# B&R Automation Studio project A2019059_Linka_Power_CP (part 37)

#### Main.st - Init, cyclic, exit code
```iecst
PROGRAM _INIT
    TprazdnyZasobnik.PT:=T#2000ms;
    TakumulaciaPlna.PT:=T#1000ms;
    TvytvorenieVakua.PT:=T#200ms;
    TodvetranieVakua.PT:=T#1s;
    TprefukPredBrzdou.PT:=T#2000ms;
    TprefukZaBrzdou.PT:=T#2000ms;
    TvysuvanieSpindle.PT:=T#1s;
    TpripravaSkrutky.PT:=T#3000ms;
    ToddelovacZakladnaPoloha.PT:=T#1000ms;
    TodsatieNecistot.PT:=T#1000ms;
    Tvibrovanie.PT:=T#3000ms;
    TvyfukovaniePredVibrovanim.PT:= T#1000ms;
    TpodaniaSkrutky.PT:= T#1000ms;
    TpredSkrutkaPripravena.PT:= T#1000ms;
    TvypnutieOfuku.PT:= T#2000ms;
    TalarmuVysunutiaSkrutkovacky.PT:= T#10s;
END_PROGRAM

PROGRAM _CYCLIC

	(********************Mapovanie IN/OUT********************************)

    SkrutkovaciSet.Manual:= P3_Srobovanie.SkrutkovaciSet_K40.Manual;
    SkrutkovaciSet.Automat:= P3_Srobovanie.SkrutkovaciSet_K40.Automat;
    SkrutkovaciSet.SkrutkaOdobrata:=P3_Srobovanie.SkrutkovaciSet_K40.SkrutkaK40_Odobrata;
    P3_Srobovanie.SkrutkovaciSet_K40.SkrutkaK40_Pripravena:= SkrutkovaciSet.SkrutkaPripravena;
    P3_Srobovanie.SkrutkovaciSet_K40.CistenieUkoncene:= SkrutkovaciSet.CistenieVykonane;
    SkrutkovaciSet.VykonajCistenie:= P3_Srobovanie.SkrutkovaciSet_K40.Cistenie;

    SkrutkovaciSet.Vreteno.IN.BrakeClosed:=P3_Srobovanie.IN.SkrutkK40_Cist_BrzdaZatvor_MS54;
    SkrutkovaciSet.Vreteno.IN.BrakeOpen:=P3_Srobovanie.IN.SkrutkK40_Cist_BrzdaOtvor_MS53;
    SkrutkovaciSet.Vreteno.IN.DeptControl:=P3_Srobovanie.IN.SkrutkK40_ZASUNUTY_MS52;
    SkrutkovaciSet.Vreteno.IN.ScrewMeasurement:=P3_Srobovanie.IN.SkrutkK40_SrobaPresla_IS81;
    SkrutkovaciSet.Vreteno.IN.ScrewMeasurementBrake:=P3_Srobovanie.IN.SkrutkK40_Cist_SrobaPresla_IS82;

    IF P3_Srobovanie.SkrutkovaciSet_K40.Reset AND SkrutkovaciSet.VretenoFaza <> 102 AND SkrutkovaciSet.VretenoFaza <> 104 THEN
        SkrutkovaciSet.VretenoFaza:=0;
        P3_Srobovanie.SkrutkovaciSet_K40.Reset:= FALSE;
    END_IF

    SkrutkovaciSet.Zasobnik.IN.AccumulationSwitch:=P3_Srobovanie.IN.ZasobSrobK40_ListaPLNA_OS15;
    SkrutkovaciSet.Zasobnik.IN.FeederLevelControl:=P3_Srobovanie.IN.ZasobSrobK40_PRAZDNY_IS79;
    SkrutkovaciSet.Zasobnik.IN.ScrewMeasurement:=P3_Srobovanie.IN.NastrelSrobK40_SrobaPresla_IS80;

    P3_Srobovanie.OUT.SkrutkK40_Cist_POSUN_YV124:=SkrutkovaciSet.Vreteno.OUT.BlastAirBrake;
    P3_Srobovanie.OUT.SkrutkK40_Cist_OTVOR_YV121:=SkrutkovaciSet.Vreteno.OUT.BrakeSpindle;
    P3_Srobovanie.OUT.SkrutkK40_OfukVakua_RUN_YV119:=SkrutkovaciSet.Vreteno.OUT.CounterBlast;
    IF SkrutkovaciSet.VretenoFaza>1 AND SkrutkovaciSet.VretenoFaza<100 THEN
        P3_Srobovanie.OUT.SkrutkK40_VYSUN_YV118:=SkrutkovaciSet.Vreteno.OUT.Spindle;
    END_IF
    P3_Srobovanie.OUT.SkrutkK40_Cist_ODSAVANIE_YV122:=SkrutkovaciSet.Vreteno.OUT.WasteExtraction;
    IF SkrutkovaciSet.VykonajCistenie THEN
        P3_Srobovanie.OUT.SkrutkK40_PrisavSkrut_RUN_YV120:=SkrutkovaciSet.Vreteno.OUT.Vacuum;
    END_IF
    P3_Srobovanie.OUT.ZasobSrobK40_Ofuk_RUN_YV114:=SkrutkovaciSet.Zasobnik.OUT.BlowOff;
    P3_Srobovanie.OUT.NastrelSrobK40_PosunSrobu_YV116:=SkrutkovaciSet.Zasobnik.OUT.Escapement;
    P3_Srobovanie.OUT.NastrelSrobK40_NastrelSrob_YV117:=SkrutkovaciSet.Zasobnik.OUT.FeedAir;
    P3_Srobovanie.OUT.ZasobSrobK40_OfukTried_RUN_YV115:=SkrutkovaciSet.Zasobnik.OUT.SortingAir;
    P3_Srobovanie.OUT.ZasobSrobK40_Vibrovanie_RUN_FM15:= SkrutkovaciSet.Zasobnik.OUT.StartA20;
    (********************Časáky********************************)
    TprazdnyZasobnik();
    TakumulaciaPlna();
    TvytvorenieVakua();
    TodvetranieVakua();
    TprefukPredBrzdou();
    TprefukZaBrzdou();
    TvysuvanieSpindle();
    TpripravaSkrutky();
    ToddelovacZakladnaPoloha();
    TodsatieNecistot();
    Tvibrovanie();
    TvyfukovaniePredVibrovanim();
    TpodaniaSkrutky();
    TpredSkrutkaPripravena();
    TvypnutieOfuku();
    TalarmuVysunutiaSkrutkovacky();
    (********************Zásobnik********************************)

    //kontrola akumulacie
    IF SkrutkovaciSet.Zasobnik.IN.AccumulationSwitch=1 THEN
        TakumulaciaPlna.IN:=1;
    ELSE
        TakumulaciaPlna.IN:=0;
    END_IF

    //kontrola naplnenia zasobnika
    IF SkrutkovaciSet.Zasobnik.IN.FeederLevelControl=1 THEN
        TprazdnyZasobnik.IN:=1;
    ELSE
        TprazdnyZasobnik.IN:=0;
    END_IF

    //Ovládanie vzduchov zásobníka//
    IF ZapniHrniec THEN
        IF TakumulaciaPlna.Q=1 THEN
            SkrutkovaciSet.Zasobnik.OUT.BlowOff:=1;
        ELSE
            SkrutkovaciSet.Zasobnik.OUT.BlowOff:=0;
        END_IF
        SkrutkovaciSet.Zasobnik.OUT.SortingAir:= 1;
    ELSE
        SkrutkovaciSet.Zasobnik.OUT.BlowOff:=0;
    END_IF

    IF NOT SkrutkovaciSet.Zasobnik.OUT.StartA20 AND NOT ZapniHrniec THEN
        TvypnutieOfuku.IN:= 1;
    ELSE
        TvypnutieOfuku.IN:= 0;
    END_IF

    IF EDGEPOS(TvypnutieOfuku.Q) THEN
        SkrutkovaciSet.Zasobnik.OUT.SortingAir:= 0;
    END_IF

    //ovladanie vibracneho podavaca
    IF ZapniHrniec THEN
        TvyfukovaniePredVibrovanim.IN:= 1;
    ELSE
        TvyfukovaniePredVibrovanim.IN:= 0;
    END_IF

    IF ZapniHrniec AND TvyfukovaniePredVibrovanim.Q THEN
        SkrutkovaciSet.Zasobnik.OUT.StartA20:=1;
        Tvibrovanie.IN:=1;
    ELSE
        SkrutkovaciSet.Zasobnik.OUT.StartA20:=0;
        Tvibrovanie.IN:=0;
    END_IF

    IF Tvibrovanie.Q=1 AND NOT P3_Srobovanie.RR_ZapniHrniec_K40 THEN
        IF TakumulaciaPlna.Q=1 THEN
            ZapniHrniec:= 0;
        END_IF
    END_IF

    //Zapnutie hrnca v ručnom režime//
    IF EDGEPOS(P3_Srobovanie.RR_ZapniHrniec_K40) THEN
        ZapniHrniec:= TRUE;
    END_IF
    IF EDGENEG(P3_Srobovanie.RR_ZapniHrniec_K40) THEN
        ZapniHrniec:= FALSE;
    END_IF

    //Zrušenie signálu skrutka pripravená//
    IF SkrutkovaciSet.SkrutkaPripravena=1 THEN
        IF SkrutkovaciSet.SkrutkaOdobrata=1 THEN
            SkrutkovaciSet.SkrutkaPripravena:=0;
        END_IF
    END_IF

    (********************Vreteno********************************)
    CASE SkrutkovaciSet.VretenoFaza OF
        0: SkrutkovaciSet.VretenoStatus:="Vypnute";
            SkrutkovaciSet.Vreteno.OUT.BlastAirBrake:=0;
            SkrutkovaciSet.Vreteno.OUT.BrakeSpindle:=0;
            SkrutkovaciSet.Vreteno.OUT.CounterBlast:=0;
            SkrutkovaciSet.Vreteno.OUT.Spindle:=0;
            SkrutkovaciSet.Vreteno.OUT.Vacuum:=0;
            SkrutkovaciSet.Vreteno.OUT.WasteExtraction:=0;

            SkrutkovaciSet.Zasobnik.OUT.Escapement:=0;
            SkrutkovaciSet.Zasobnik.OUT.FeedAir:=0;

            SkrutkovaciSet.Zasobnik.OUT.StartA20:=0;

            SkrutkovaciSet.CistenieVykonane:=0;
            SkrutkovaciSet.SkrutkaPripravena:=0;

            TprazdnyZasobnik.IN:=0;
            TakumulaciaPlna.IN:=0;
            TvytvorenieVakua.IN:=0;
            TodvetranieVakua.IN:=0;
            TprefukPredBrzdou.IN:=0;
            TprefukZaBrzdou.IN:=0;
            TvysuvanieSpindle.IN:=0;
            TpripravaSkrutky.IN:=0;
            ToddelovacZakladnaPoloha.IN:=0;
            TodsatieNecistot.IN:=0;
            TpodaniaSkrutky.IN:= 0;
            TpredSkrutkaPripravena.IN:= 0;
            ZapniHrniec:= 0;
            PocetPokusovOpripravuSkrutky:=0;
            TalarmuVysunutiaSkrutkovacky.IN:= 0;
            StavSkrutkovackaVysunuta:= 0;
            SkrutkovaciSet.VretenoFaza:=1;

        1: SkrutkovaciSet.VretenoStatus:="Inicializacia: cakam na povel";
            IF SkrutkovaciSet.Automat=1 THEN
                SkrutkovaciSet.CistenieVykonane:=0;
                SkrutkovaciSet.SkrutkaPripravena:=0;
                SkrutkovaciSet.VretenoFaza:=2;
            ELSIF SkrutkovaciSet.Manual=1 THEN
                SkrutkovaciSet.VretenoFaza:=250;
            END_IF

        2: SkrutkovaciSet.VretenoStatus:="Inicializacia: cakam na povel precisti hadice";

            IF SkrutkovaciSet.VykonajCistenie=1 THEN
                SkrutkovaciSet.Vreteno.OUT.Vacuum:=1;
                SkrutkovaciSet.VretenoFaza:=3;
            END_IF

        3: SkrutkovaciSet.VretenoStatus:="Inicializacia: Cakam na snimac: vreteno vysunute";
            SkrutkovaciSet.Vreteno.OUT.Spindle:=1;
            TalarmuVysunutiaSkrutkovacky.IN:= 1;

            IF P3_Srobovanie.IN.SkrutkK40_VysunutieHrotu_IOS11 > 1 THEN
                StavSkrutkovackaVysunuta:= TRUE;
                TvysuvanieSpindle.IN:=1;
            END_IF

            IF TvysuvanieSpindle.Q=1 AND StavSkrutkovackaVysunuta THEN
                TodvetranieVakua.IN:= 1;
                SkrutkovaciSet.Vreteno.OUT.CounterBlast:=1;
                SkrutkovaciSet.Vreteno.OUT.Vacuum:=0;
            END_IF

            IF TvysuvanieSpindle.Q AND StavSkrutkovackaVysunuta AND TodvetranieVakua.Q THEN
                StavSkrutkovackaVysunuta:= FALSE;
                TalarmuVysunutiaSkrutkovacky.IN:= 0;
                TvysuvanieSpindle.IN:=0;
                TodvetranieVakua.IN:= 0;
                SkrutkovaciSet.VretenoFaza:=4;
            ELSIF TalarmuVysunutiaSkrutkovacky.Q THEN
                P34_Alarmy[342]:= TRUE;
                P3_PoruchaST1:= TRUE;
            END_IF

        4: SkrutkovaciSet.VretenoStatus:="Inicializacia: Cakam na snimac: vreteno zasunute";
            SkrutkovaciSet.Vreteno.OUT.Spindle:=0;
            IF SkrutkovaciSet.Vreteno.IN.DeptControl=1 THEN
                SkrutkovaciSet.Vreteno.OUT.CounterBlast:=0;
                SkrutkovaciSet.VretenoFaza:=5;
            END_IF

        5: SkrutkovaciSet.VretenoStatus:="Inicializacia: Cakam na prefuknutie hadice za brzdou";
            TprefukZaBrzdou.IN:=1;
            SkrutkovaciSet.Vreteno.OUT.BlastAirBrake:=1;
            IF TprefukZaBrzdou.Q=1 THEN
                TprefukZaBrzdou.IN:=0;
                SkrutkovaciSet.Vreteno.OUT.BlastAirBrake:=0;
                SkrutkovaciSet.VretenoFaza:=6;
            END_IF

        6: SkrutkovaciSet.VretenoStatus:="Inicializacia: vypinam prefuk";
            TprefukZaBrzdou.IN:=0;
            SkrutkovaciSet.Vreteno.OUT.BlastAirBrake:=0;
            SkrutkovaciSet.Vreteno.OUT.Vacuum:=1;
            SkrutkovaciSet.VretenoFaza:=7;

        7: SkrutkovaciSet.VretenoStatus:="Inicializacia: Cakam na snimac: vreteno vysunute";
            SkrutkovaciSet.Vreteno.OUT.Spindle:=1;
            TalarmuVysunutiaSkrutkovacky.IN:= 1;

            IF P3_Srobovanie.IN.SkrutkK40_VysunutieHrotu_IOS11 > 1 THEN
                StavSkrutkovackaVysunuta:= TRUE;
                TvysuvanieSpindle.IN:=1;
            END_IF

            IF TvysuvanieSpindle.Q=1 AND StavSkrutkovackaVysunuta THEN
                TodvetranieVakua.IN:= 1;
                SkrutkovaciSet.Vreteno.OUT.CounterBlast:=1;
                SkrutkovaciSet.Vreteno.OUT.Vacuum:=0;
            END_IF

            IF TvysuvanieSpindle.Q AND StavSkrutkovackaVysunuta AND TodvetranieVakua.Q THEN
                StavSkrutkovackaVysunuta:= FALSE;
                TalarmuVysunutiaSkrutkovacky.IN:= 0;
                TvysuvanieSpindle.IN:=0;
                TodvetranieVakua.IN:= 0;
                SkrutkovaciSet.VretenoFaza:=8;
            ELSIF TalarmuVysunutiaSkrutkovacky.Q THEN
                P34_Alarmy[342]:= TRUE;
                P3_PoruchaST1:= TRUE;
            END_IF

        8: SkrutkovaciSet.VretenoStatus:="Inicializacia: Cakam na snimac: vreteno zasunute";
            SkrutkovaciSet.Vreteno.OUT.Spindle:=0;
            IF SkrutkovaciSet.Vreteno.IN.DeptControl=1 THEN
                SkrutkovaciSet.Vreteno.OUT.CounterBlast:=0;
                SkrutkovaciSet.VretenoFaza:=9;
            END_IF

        9: SkrutkovaciSet.VretenoStatus:="Inicializacia: Cakam na prefuknutie hadice pred brzdou";
            TprefukPredBrzdou.IN:=1;
            SkrutkovaciSet.Zasobnik.OUT.FeedAir:=1;
            IF TprefukPredBrzdou.Q=1 THEN
                TprefukPredBrzdou.IN:=0;
                SkrutkovaciSet.Zasobnik.OUT.FeedAir:=0;
                SkrutkovaciSet.VretenoFaza:=10;
            END_IF

        10: SkrutkovaciSet.VretenoStatus:="Inicializacia: Cakam na snimac: brzda uvolnena";
            SkrutkovaciSet.Vreteno.OUT.BrakeSpindle:=1;
            IF SkrutkovaciSet.Vreteno.IN.BrakeOpen=1 THEN
                SkrutkovaciSet.Vreteno.OUT.BlastAirBrake:=1;
                SkrutkovaciSet.VretenoFaza:=11;
            END_IF

        11: SkrutkovaciSet.VretenoStatus:="Inicializacia: Cakam na prefuknutie hadice za brzdou";
            TprefukZaBrzdou.IN:=1;
            SkrutkovaciSet.Vreteno.OUT.BlastAirBrake:=1;
            IF TprefukZaBrzdou.Q=1 THEN
                TprefukZaBrzdou.IN:=0;
                SkrutkovaciSet.Vreteno.OUT.BlastAirBrake:=0;
                SkrutkovaciSet.VretenoFaza:=12;
            END_IF

        12: SkrutkovaciSet.VretenoStatus:="Inicializacia: vypinam prefuk";
            TprefukZaBrzdou.IN:=0;
            SkrutkovaciSet.Vreteno.OUT.BlastAirBrake:=0;
            SkrutkovaciSet.Vreteno.OUT.Vacuum:=1;
            SkrutkovaciSet.VretenoFaza:=13;

        13: SkrutkovaciSet.VretenoStatus:="Inicializacia: Cakam na snimac: vreteno vysunute";
            SkrutkovaciSet.Vreteno.OUT.Spindle:=1;
            TalarmuVysunutiaSkrutkovacky.IN:= 1;

            IF P3_Srobovanie.IN.SkrutkK40_VysunutieHrotu_IOS11 > 1 THEN
                StavSkrutkovackaVysunuta:= TRUE;
                TvysuvanieSpindle.IN:=1;
            END_IF

            IF TvysuvanieSpindle.Q=1 AND StavSkrutkovackaVysunuta THEN
                TodvetranieVakua.IN:= 1;
                SkrutkovaciSet.Vreteno.OUT.CounterBlast:=1;
                SkrutkovaciSet.Vreteno.OUT.Vacuum:=0;
            END_IF

            IF TvysuvanieSpindle.Q AND StavSkrutkovackaVysunuta AND TodvetranieVakua.Q THEN
                StavSkrutkovackaVysunuta:= FALSE;
                TalarmuVysunutiaSkrutkovacky.IN:= 0;
                TvysuvanieSpindle.IN:=0;
                TodvetranieVakua.IN:= 0;
                SkrutkovaciSet.VretenoFaza:=14;
            ELSIF TalarmuVysunutiaSkrutkovacky.Q THEN
                P34_Alarmy[342]:= TRUE;
                P3_PoruchaST1:= TRUE;
            END_IF

        14: SkrutkovaciSet.VretenoStatus:="Inicializacia: Cakam na snimac: vreteno zasunute";
            SkrutkovaciSet.Vreteno.OUT.Spindle:=0;
            IF SkrutkovaciSet.Vreteno.IN.DeptControl=1 THEN
                SkrutkovaciSet.Vreteno.OUT.CounterBlast:=0;
                SkrutkovaciSet.VretenoFaza:=15;
            END_IF

        15: SkrutkovaciSet.VretenoStatus:="Inicializacia: Cakam na snimac: brzda zasunuta";
            SkrutkovaciSet.Vreteno.OUT.BrakeSpindle:=0;
            IF SkrutkovaciSet.Vreteno.IN.BrakeClosed=1 THEN
                SkrutkovaciSet.CistenieVykonane:=1;
                SkrutkovaciSet.VretenoFaza:=16;
            END_IF

        16: SkrutkovaciSet.VretenoStatus:="Inicializacia: Cakam na zrusenie signalu: vykonaj cistenie";
            IF SkrutkovaciSet.VykonajCistenie=0 THEN
                SkrutkovaciSet.CistenieVykonane:=0;
                SkrutkovaciSet.SkrutkaPripravena:=0;
                SkrutkovaciSet.VretenoFaza:=100;
            END_IF

        100: SkrutkovaciSet.VretenoStatus:="Cakam kym zasobnik pripravy skrutku";
            ZapniHrniec:= 1;
            IF TakumulaciaPlna.Q=1 AND SkrutkovaciSet.Zasobnik.OUT.StartA20 THEN
                TpodaniaSkrutky.IN:= 1;
            END_IF

            IF TpodaniaSkrutky.Q THEN
                TpodaniaSkrutky.IN:= 0;
                SkrutkovaciSet.VretenoFaza:=102;
            END_IF

        102: SkrutkovaciSet.VretenoStatus:="Cakam na snimac: skrutka presla hadicou";
            SkrutkovaciSet.Zasobnik.OUT.Escapement:=1;
            TpripravaSkrutky.IN:=1;
            IF SkrutkovaciSet.Zasobnik.IN.ScrewMeasurement=1 THEN
                SkrutkovaciSet.Zasobnik.OUT.FeedAir:=1;
                TpripravaSkrutky.IN:=0;
                SkrutkovaciSet.VretenoFaza:=104;
            ELSIF TpripravaSkrutky.Q=1 THEN
                TpripravaSkrutky.IN:=0;
                SkrutkovaciSet.Zasobnik.OUT.Escapement:=0;
                SkrutkovaciSet.VretenoFaza:=100;
            END_IF

        104: SkrutkovaciSet.VretenoStatus:="Cakam na snimac: skrutka presla hadicou pred brzdou";
            IF SkrutkovaciSet.Vreteno.IN.ScrewMeasurementBrake=1 THEN
                SkrutkovaciSet.Zasobnik.OUT.Escapement:=0;
                SkrutkovaciSet.Zasobnik.OUT.FeedAir:=0;
                PocetPokusovOpripravuSkrutky:=0;
                SkrutkovaciSet.VretenoFaza:=106;
            END_IF

        106: SkrutkovaciSet.VretenoStatus:="Cakam na odsatie necistot";
            SkrutkovaciSet.Vreteno.OUT.WasteExtraction:=1;
            TodsatieNecistot.IN:=1;
            IF TodsatieNecistot.Q=1 THEN
                TodsatieNecistot.IN:=0;
                SkrutkovaciSet.Vreteno.OUT.WasteExtraction:=0;
                SkrutkovaciSet.VretenoFaza:=107;
            END_IF

        107: SkrutkovaciSet.VretenoStatus:="Cakam kym skrutkovacka odoberie skrutku";
            IF SkrutkovaciSet.SkrutkaPripravena=0 AND SkrutkovaciSet.SkrutkaOdobrata=0 THEN
                SkrutkovaciSet.VretenoFaza:=108;
            END_IF

        108: SkrutkovaciSet.VretenoStatus:="Cakam na snimac: brzda uvolnena";
            SkrutkovaciSet.Vreteno.OUT.BrakeSpindle:=1;
            IF SkrutkovaciSet.Vreteno.IN.BrakeOpen=1 THEN
                SkrutkovaciSet.Vreteno.OUT.BlastAirBrake:=1;
                SkrutkovaciSet.VretenoFaza:=110;
            END_IF

        110: SkrutkovaciSet.VretenoStatus:="Cakam na snimac: skrutka presla hadicou pred vretenom";
            IF SkrutkovaciSet.Vreteno.IN.ScrewMeasurement=1 THEN
                SkrutkovaciSet.Vreteno.OUT.BlastAirBrake:=0;
                SkrutkovaciSet.Vreteno.OUT.BrakeSpindle:=0;
                SkrutkovaciSet.VretenoFaza:=112;
            END_IF

        112: SkrutkovaciSet.VretenoStatus:="Cakam na snimac: brzda zabrzdena";
            SkrutkovaciSet.Vreteno.OUT.BrakeSpindle:=0;
            IF SkrutkovaciSet.Vreteno.IN.BrakeClosed=1 AND SkrutkovaciSet.SkrutkaOdobrata=0 THEN
                TpredSkrutkaPripravena.IN:= 1;
                IF TpredSkrutkaPripravena.Q THEN
                    TpredSkrutkaPripravena.IN:= 0;
                    SkrutkovaciSet.SkrutkaPripravena:=1;
                    SkrutkovaciSet.VretenoFaza:=100;
                END_IF
            END_IF

            //*************** opakovany pokus o oddelenie skrutky *********************************

        170: SkrutkovaciSet.VretenoStatus:="Cakam na presunutie oddelovaca do zakladnej polohy";
            SkrutkovaciSet.Zasobnik.OUT.Escapement:=0;
            ToddelovacZakladnaPoloha.IN:=1;
            IF ToddelovacZakladnaPoloha.Q=1 THEN
                ToddelovacZakladnaPoloha.IN:=0;
                PocetPokusovOpripravuSkrutky:=PocetPokusovOpripravuSkrutky+1;
                IF PocetPokusovOpripravuSkrutky>3 THEN
                    PocetPokusovOpripravuSkrutky:=0;
                    SkrutkovaciSet.VretenoFaza:=171;
                ELSE
                    SkrutkovaciSet.VretenoFaza:=100;
                END_IF
            END_IF

        171: SkrutkovaciSet.VretenoStatus:="Zaseknuta skrutka v oddelovaci!!!";

    END_CASE
END_PROGRAM

PROGRAM _EXIT
END_PROGRAM
```

#### Types.typ - Local data types
```iecst
TYPE
	SkrutkovaciSetStruc1 : 	STRUCT
		VretenoStatus : WSTRING[80];
		VretenoFaza : USINT;
		Zasobnik : ZasobnikStruc;
		Vreteno : VretenoStruc;
		SkrutkaOdobrata : BOOL;
		SkrutkaPripravena : BOOL;
		Manual : BOOL;
		PodajSrobu : BOOL;
		CistenieVykonane : BOOL;
		VykonajCistenie : BOOL;
		Automat : BOOL;
	END_STRUCT;
	INzasobnik1 : 	STRUCT
		AccumulationSwitch : BOOL; (*Snimac zaplnenia S25*)
		ScrewMeasurement : BOOL; (*Kontrola matice S21*)
		FeederLevelControl : BOOL; (*Hladina v zasobniku S20*)
	END_STRUCT;
	OUTzasobnik1 : 	STRUCT
		StartA20 : BOOL; (*Zapnutie vibrovania A20*)
		Escapement : BOOL; (*Pustanie matky do hadice Y22*)
		FeedAir : BOOL; (*Strielanie do hadice Y21*)
		SortingAir : BOOL; (*Triedenie kusov Y30*)
		BlowOff : BOOL; (*Zhadzovanie kusov Y25*)
	END_STRUCT;
	INvreteno1 : 	STRUCT
		ReturnStroke : BOOL; (*Vreteno zasunute S01*)
		DeptControl : BOOL; (*Vreteno vysunute S02*)
		BrakeClosed : BOOL; (*Brzda zatvorena S13*)
		BrakeOpen : BOOL; (*Brzda otvorena S12*)
		ScrewMeasurementBrake : BOOL; (*Kontrola matice pred brzdou S15*)
		ScrewMeasurement : BOOL; (*Kontrola matice v hadici S06*)
	END_STRUCT;
	OUTvreteno1 : 	STRUCT
		WasteExtraction : BOOL; (*Odstranovanie spiny Y13*)
		Spindle : BOOL; (*Vysunutie vretena Y02*)
		BlastAirBrake : BOOL; (*Strielanie za brzdou Y14*)
		BrakeSpindle : BOOL; (*Brzda vretena Y12*)
		Vacuum : BOOL; (*Pridrzanie skrutky Y15*)
		CounterBlast : BOOL; (*Uvolnenie skrutky Y16*)
	END_STRUCT;
	VretenoStruc1 : 	STRUCT
		OUT : OUTvreteno;
		IN : INvreteno;
	END_STRUCT;
	ZasobnikStruc1 : 	STRUCT
		OUT : OUTzasobnik;
		IN : INzasobnik;
	END_STRUCT;
	SkrutkovaciSetStruc : 	STRUCT
		VretenoStatus : WSTRING[80];
		VretenoFaza : USINT;
		Zasobnik : ZasobnikStruc;
		Vreteno : VretenoStruc;
		SkrutkaOdobrata : BOOL;
		SkrutkaPripravena : BOOL;
		Manual : BOOL;
		PodajSrobu : BOOL;
		CistenieVykonane : BOOL;
		VykonajCistenie : BOOL;
		Automat : BOOL;
	END_STRUCT;
	INzasobnik : 	STRUCT
		AccumulationSwitch : BOOL; (*Snimac zaplnenia S25*)
		ScrewMeasurement : BOOL; (*Kontrola matice S21*)
		FeederLevelControl : BOOL; (*Hladina v zasobniku S20*)
	END_STRUCT;
	OUTzasobnik : 	STRUCT
		StartA20 : BOOL; (*Zapnutie vibrovania A20*)
		Escapement : BOOL; (*Pustanie matky do hadice Y22*)
		FeedAir : BOOL; (*Strielanie do hadice Y21*)
		SortingAir : BOOL; (*Triedenie kusov Y30*)
		BlowOff : BOOL; (*Zhadzovanie kusov Y25*)
	END_STRUCT;
	INvreteno : 	STRUCT
		ReturnStroke : BOOL; (*Vreteno zasunute S01*)
		DeptControl : BOOL; (*Vreteno vysunute S02*)
		BrakeClosed : BOOL; (*Brzda zatvorena S13*)
		BrakeOpen : BOOL; (*Brzda otvorena S12*)
		ScrewMeasurementBrake : BOOL; (*Kontrola matice pred brzdou S15*)
		ScrewMeasurement : BOOL; (*Kontrola matice v hadici S06*)
	END_STRUCT;
	OUTvreteno : 	STRUCT
		WasteExtraction : BOOL; (*Odstranovanie spiny Y13*)
		Spindle : BOOL; (*Vysunutie vretena Y02*)
		BlastAirBrake : BOOL; (*Strielanie za brzdou Y14*)
		BrakeSpindle : BOOL; (*Brzda vretena Y12*)
		Vacuum : BOOL; (*Pridrzanie skrutky Y15*)
		CounterBlast : BOOL; (*Uvolnenie skrutky Y16*)
	END_STRUCT;
	VretenoStruc : 	STRUCT
		OUT : OUTvreteno;
		IN : INvreteno;
	END_STRUCT;
	ZasobnikStruc : 	STRUCT
		OUT : OUTzasobnik;
		IN : INzasobnik;
	END_STRUCT;
END_TYPE
```

#### Variables.var - Local variables
```iecst
VAR
	SkrutkovaciSet : SkrutkovaciSetStruc;
	TprazdnyZasobnik : TON;
	TakumulaciaPlna : TON;
	TvytvorenieVakua : TON;
	TodvetranieVakua : TON;
	TprefukPredBrzdou : TON;
	TvysuvanieSpindle : TON;
	TprefukZaBrzdou : TON;
	PocetPokusovOpripravuSkrutky : USINT;
	ToddelovacZakladnaPoloha : TON;
	TpripravaSkrutky : TON;
	TodsatieNecistot : TON;
	Tvibrovanie : TON;
	TvyfukovaniePredVibrovanim : TON;
	ZapniHrniec : BOOL;
	TpodaniaSkrutky : TON;
	TpredSkrutkaPripravena : TON;
	TvypnutieOfuku : TON;
	StavSkrutkovackaVysunuta : BOOL;
	TalarmuVysunutiaSkrutkovacky : TON;
END_VAR
```

### Program Logical/Program/Pracovisko_3/P3_AkumulacnyStoper (IEC)

#### Main.st - Init, cyclic, exit code
```iecst
PROGRAM _INIT
	(* Insert code here *)

END_PROGRAM

PROGRAM _CYCLIC

	//Volanie funkcie SequenceControl//
    SequenceControl(SC:= SC_P3_AkumulacnyStoper);

    //Reset sekcie //
    IF NOT Safety.STAV.P3_ZonaBunky_AKTIVNA THEN
        SC_P3_AkumulacnyStoper.Step:= 0;
    ELSIF P3_AkumulacnyStoper.Reset THEN
        SC_P3_AkumulacnyStoper.Step:= 0;
        P3_AkumulacnyStoper.Reset:= FALSE;
    END_IF

    CASE SC_P3_AkumulacnyStoper.Step OF

        0:
            SC_P3_AkumulacnyStoper.StepName:='0 - Nulovanie';
            P3_AkumulacnyStoper.Automat:= FALSE;
            P3_AkumulacnyStoper.KoniecCyklu:= FALSE;
            P3_AkumulacnyStoper.Manual:= FALSE;
            P3_AkumulacnyStoper.STAV.PoINIT:= FALSE;
            P3_AkumulacnyStoper.OUT.ZasunStoper_YV133:= FALSE;
			P3_AkumulacnyStoper.STAV.PrebiehaVyvezeniePaletky:= FALSE;

            IF Safety.STAV.P3_ZonaBunky_AKTIVNA AND NOT P3_Pracovisko.STAV.PORUCHA AND P3_Pracovisko.IN.PrivodVzduchu_SnimacTlaku_S25 THEN
                SC_P3_AkumulacnyStoper.ResetStep:= TRUE;
                SC_P3_AkumulacnyStoper.Step:= 1;
            END_IF

        1:
            SC_P3_AkumulacnyStoper.StepName:='1 - Cakam na spustenie vyroby';
            P3_AkumulacnyStoper.KoniecCyklu:= FALSE;
            IF P3_AkumulacnyStoper.Automat THEN
                SC_P3_AkumulacnyStoper.Step:= 2;
            ELSIF P3_AkumulacnyStoper.Manual THEN
                SC_P3_AkumulacnyStoper.Step:= 700;
            END_IF

            //********************************************************Inicializácia****************************************************************************//
        2:
            SC_P3_AkumulacnyStoper.StepName:='2 - Inicializacia - cakam na spustenie inicializacie';
            SC_P3_AkumulacnyStoper.IdleTime.PT:= T#4s;
            SC_P3_AkumulacnyStoper.AlarmTime.PT:= T#5s;

            IF P3_Dopravniky.STAV.PoINIT THEN
                SC_P3_AkumulacnyStoper.ResetStep:= TRUE;
                SC_P3_AkumulacnyStoper.Step:= 3;
            END_IF

        3:
            SC_P3_AkumulacnyStoper.StepName:='3 - Inicializacia - hladanie paletky';
            SC_P3_AkumulacnyStoper.IdleTime.PT:= T#5s;
            SC_P3_AkumulacnyStoper.AlarmTime.PT:= T#5s;
            SC_P3_AkumulacnyStoper.IdleTime.IN:= TRUE;

            IF P3_AkumulacnyStoper.IN.PritomnPaletky_IS65 THEN
                P3_AkumulacnyStoper.STAV.PoINIT:= TRUE;
                SC_P3_AkumulacnyStoper.ResetStep:= TRUE;
                SC_P3_AkumulacnyStoper.Step:= 101;
            ELSIF SC_P3_AkumulacnyStoper.IdleTime.Q THEN
                P3_AkumulacnyStoper.STAV.PoINIT:= TRUE;
                SC_P3_AkumulacnyStoper.ResetStep:= TRUE;
                SC_P3_AkumulacnyStoper.Step:= 100;
            END_IF

            //********************************************************Automatický režim****************************************************************************//
        100:
            SC_P3_AkumulacnyStoper.StepName:='100 - Automaticky Rezim - cakam na príchod paletky na stoper';
            SC_P3_AkumulacnyStoper.IdleTime.PT:= T#200ms;
            SC_P3_AkumulacnyStoper.AlarmTime.PT:= T#5s;

            IF P3_AkumulacnyStoper.IN.PritomnPaletky_IS65 THEN
                P3_StoperSrobovania.STAV.PrebiehaVyvezeniePaletky:= FALSE;
            END_IF

            SC_P3_AkumulacnyStoper.IdleTime.IN:= P3_AkumulacnyStoper.IN.PritomnPaletky_IS65;

            IF P3_AkumulacnyStoper.KoniecCyklu THEN
                SC_P3_AkumulacnyStoper.ResetStep:= TRUE;
                SC_P3_AkumulacnyStoper.Step:= 0;
            ELSIF SC_P3_AkumulacnyStoper.IdleTime.Q THEN
                SC_P3_AkumulacnyStoper.ResetStep:= TRUE;
                SC_P3_AkumulacnyStoper.Step:= 101;
            END_IF

        101:
            SC_P3_AkumulacnyStoper.StepName:='101 - Automaticky Rezim - cakam na vyvezenie paletky na stoper Leakage test A';
            SC_P3_AkumulacnyStoper.IdleTime.PT:= T#200ms;
            SC_P3_AkumulacnyStoper.AlarmTime.PT:= T#5s;

            IF P3_AkumulacnyStoper.KoniecCyklu THEN
                SC_P3_AkumulacnyStoper.ResetStep:= TRUE;
                SC_P3_AkumulacnyStoper.Step:= 0;
            ELSIF ((SC_P3_LeakageTestA.Step = 100 AND NOT P3_LeakageTestA.IN.PritomnostPaletky_S23) OR (P3_LeakageTestA.OUT.ZasunStoper_YV134 AND SC_P3_LeakageTestA.Step = 561)) AND NOT P3_AkumulacnyStoper.STAV.PrebiehaVyvezeniePaletky THEN
                SC_P3_AkumulacnyStoper.ResetStep:= TRUE;
                SC_P3_AkumulacnyStoper.Step:= 105;
            ELSIF NOT P3_AkumulacnyStoper.IN.PritomnPaletky_IS65 THEN
                SC_P3_AkumulacnyStoper.ResetStep:= TRUE;
                SC_P3_AkumulacnyStoper.Step:= 100;
            END_IF

        105:
            SC_P3_AkumulacnyStoper.StepName:='105 - Automaticky Rezim - vyvazam paletku na stoper Leakage test A';
            SC_P3_AkumulacnyStoper.IdleTime.PT:= T#200ms;
            SC_P3_AkumulacnyStoper.AlarmTime.PT:= T#10s;

            SC_P3_AkumulacnyStoper.AlarmTime.IN:= P3_AkumulacnyStoper.IN.PritomnPaletky_IS65;

            IF NOT SC_P3_AkumulacnyStoper.Switch1 THEN
                P3_AkumulacnyStoper.OUT.ZasunStoper_YV133:= TRUE;
                P3_AkumulacnyStoper.STAV.PrebiehaVyvezeniePaletky:= TRUE;
                SC_P3_AkumulacnyStoper.Switch1:= TRUE;
            END_IF

            IF NOT P3_AkumulacnyStoper.IN.PritomnPaletky_IS65 THEN
                P3_AkumulacnyStoper.OUT.ZasunStoper_YV133:= FALSE;
                SC_P3_AkumulacnyStoper.Step:= 100;
            ELSIF SC_P3_AkumulacnyStoper.AlarmTime.Q THEN
                P34_Alarmy[356]:= TRUE;
                P3_Pracovisko.KoniecCyklu:= TRUE;
                SC_P3_AkumulacnyStoper.ResetStep:= TRUE;
                SC_P3_AkumulacnyStoper.Step:= 0;
            END_IF

            //*******************************************************Manuálny režim*******************************************************************************//
        700:
            SC_P3_AkumulacnyStoper.StepName:='700 - Manualny Rezim';
            SC_P3_AkumulacnyStoper.IdleTime.PT:= T#8s;
            SC_P3_AkumulacnyStoper.AlarmTime.PT:= T#5s;

    END_CASE

END_PROGRAM

PROGRAM _EXIT
	(* Insert code here *)

END_PROGRAM
```

#### Variables.var - Local variables
```iecst
VAR
	TEST : BOOL;
END_VAR
```

### Program Logical/Program/Pracovisko_3/P3_StoperLeakageTestA (IEC)

#### Main.st - Init, cyclic, exit code
```iecst
PROGRAM _INIT
    Triger_0:= FALSE;
    Triger_1:= FALSE;

    P3_LeakageTestA.STAV.Tester_ON:= TRUE;
END_PROGRAM

PROGRAM _CYCLIC

	//Volanie podprogramov//
    OvlCentrovacky;
    IOLinkKomunikacia;
    OvlPritlaku;
    TesterKomunikacia;

    //Volanie funkcie SequenceControl//
    SequenceControl(SC:= SC_P3_LeakageTestA);

    //Príznak leakage test A východzia pozícia//
    IF P3_LeakageTestA.IN.Centrovanie_ZASUNUTE_IS72 AND P3_LeakageTestA.IN.Pritlak_ZASUNUTY_MS46 AND P3_LeakageTestA.IN.Kopito_ZASUNUTE_IS68 THEN
        P3_LeakageTestA_VychodziaPozicia:= TRUE;
    ELSE
        P3_LeakageTestA_VychodziaPozicia:= FALSE;
    END_IF

    //Reset sekcie //
    IF P3_LeakageTestA.Reset THEN
        SC_P3_LeakageTestA.Step:= 0;
        P3_LeakageTestA.Reset:= FALSE;
    END_IF

    IF NOT Safety.STAV.P3_ZonaBunky_AKTIVNA AND NOT P3_LeakageTestA.Automat THEN
        SC_P3_LeakageTestA.Step:= 0;
    END_IF

    IF NOT Safety.STAV.P3_ZonaBunky_AKTIVNA AND NOT Triger_0 THEN
        Triger_0:= TRUE;
        IF P3_LeakageTestA.IN.PritomnostPaletky_S23 AND P3_LeakageTestA.Automat THEN
            IF NOT Paletka[i].VnutornyStav.KomunikaciaOtvorena THEN
                SC_P3_LeakageTestA.ResetStep:= TRUE;
                SC_P3_LeakageTestA.Step:= 0;
            ELSIF Paletka[i].VnutornyStav.KomunikaciaUzavreta THEN
                SC_P3_LeakageTestA.ResetStep:= TRUE;
                SC_P3_LeakageTestA.Step:= 0;
            ELSIF Paletka[i].VnutornyStav.KomunikaciaOtvorena THEN
                Paletka[i].PAR.StavPowerCP:= 'FAIL';
                Paletka[i].PAR.StavPaletky:= 'NG';
                P3_LeakageTestA.KoniecCyklu:= TRUE;
                SC_P3_LeakageTestA.ResetStep:= TRUE;
                SC_P3_LeakageTestA.Step:= 550;
            END_IF
        END_IF
    END_IF

    IF Safety.STAV.P3_ZonaBunky_AKTIVNA THEN
        Triger_0:= FALSE;
    END_IF

    //Porucha stanice//
    IF P3_PoruchaST2 AND NOT Triger_1 THEN
        Triger_1:= TRUE;
        IF P3_LeakageTestA.IN.PritomnostPaletky_S23 AND P3_LeakageTestA.Automat THEN
            IF NOT Paletka[i].VnutornyStav.KomunikaciaOtvorena THEN
                SC_P3_LeakageTestA.ResetStep:= TRUE;
                SC_P3_LeakageTestA.Step:= 0;
            ELSIF Paletka[i].VnutornyStav.KomunikaciaUzavreta THEN
                SC_P3_LeakageTestA.ResetStep:= TRUE;
                SC_P3_LeakageTestA.Step:= 0;
            ELSIF Paletka[i].VnutornyStav.KomunikaciaOtvorena THEN
                Paletka[i].PAR.StavPowerCP:= 'FAIL';
                Paletka[i].PAR.StavPaletky:= 'NG';
                P3_LeakageTestA.KoniecCyklu:= TRUE;
                SC_P3_LeakageTestA.ResetStep:= TRUE;
                SC_P3_LeakageTestA.Step:= 550;
            END_IF
        ELSE
            SC_P3_LeakageTestA.ResetStep:= TRUE;
            SC_P3_LeakageTestA.Step:= 0;
        END_IF
    END_IF

    IF NOT P3_PoruchaST2 THEN
        Triger_1:= FALSE;
    END_IF

    CASE SC_P3_LeakageTestA.Step OF

        0:
            SC_P3_LeakageTestA.StepName:='0 - Nulovanie';
            SC_OvlCentrovacky.Step:= 0;
            SC_OvlPritlaku.Step:= 0;
            P3_LeakageTestA.Automat:= FALSE;
            P3_LeakageTestA.KoniecCyklu:= FALSE;
            P3_LeakageTestA.Manual:= FALSE;
            P3_LeakageTestA.STAV.PoINIT:= FALSE;
            P3_LeakageTestA.OUT.Kopito_VYSUN_YV141:= FALSE;
            P3_LeakageTestA.OUT.Kopito_ZASUN_YV142:= TRUE;
            P3_LeakageTestA.OUT.ZasunStoper_YV134:= FALSE;
            (*P3_LeakageTestA.OUT.PneuZamok_ODOMKNI_YV159:= FALSE;*)
            P3_LeakageTestA.STAV.KOM_PLC_OdoslanieFotiek_OK:= FALSE;
            P3_LeakageTestA.STAV.KOM_PLC_VymazanieFotiek_OK:= FALSE;
            TRCB_P3_LeakageTestA_ST8A.CMD.VyziadajStavPaletky_TYP1:= FALSE;
            TRCB_P3_LeakageTestA_ST8A.CMD.PriradQRkodFiltra_TYP3:= FALSE;
            TRCB_P3_LeakageTestA_ST8A.CMD.OdosliStavPaletky_TYP2:= FALSE;
            AteqLeakageTester_A.CitajParametreTestera:= FALSE;
            PrecitaneCisloPaletky:= '';
            AteqLeakageTester_A.START_Testovania:= FALSE;
            PocetDopytovNaServer:= 0;
            Taktime_LeakageTestA_ST8A.CMD.START_Merania_1:= FALSE;
            Taktime_LeakageTestA_ST8A.CMD.START_Merania_2:= FALSE;
            PaletkaPrechadza:= FALSE;
            P3_LeakageTestA.STAV.PrebiehaVyvezeniePaletky:= FALSE;
            TestovaciKus:= FALSE;
            Revork:= FALSE;
            P3_LeakageTestA.RR_TestovanieLeakageTestu:= FALSE;
            P3_LeakageTestA.RR_VysunSpodneKopito:= FALSE;
            P3_LeakageTestA.RR_TestovaciaSekvencia:= FALSE;
            P3_LeakageTestA.STAV.TestovaciaSekvencia_BUSY:= FALSE;
            PocetOpakovaniTestu:= 0;
            OpakovanyTest:= FALSE;
            P34_Vizu.ZobrazHL1_ST8:= FALSE;
            TRCB_P3_LeakTestA_OpatovnyDopyt:= FALSE;
            TRCB_P3_LeakTestA_PaletkaNG:= FALSE;

            IF Safety.STAV.P3_ZonaBunky_AKTIVNA AND NOT P3_Pracovisko.STAV.PORUCHA AND P3_Pracovisko.IN.PrivodVzduchu_SnimacTlaku_S25 THEN
                SC_P3_LeakageTestA.ResetStep:= TRUE;
                SC_P3_LeakageTestA.Step:= 1;
            END_IF

        1:
            SC_P3_LeakageTestA.StepName:='1 - Cakam na spustenie vyroby';
            P3_LeakageTestA.KoniecCyklu:= FALSE;
            IF P3_LeakageTestA.Automat THEN
                SC_P3_LeakageTestA.Step:= 2;
            ELSIF P3_LeakageTestA.Manual THEN
                SC_P3_LeakageTestA.Step:= 700;
            END_IF

            //********************************************************Inicializácia****************************************************************************//

        2:
            SC_P3_LeakageTestA.StepName:='2 - Inicializacia - cakam na spustenie inicializacie';
            SC_P3_LeakageTestA.IdleTime.PT:= T#2s;
            SC_P3_LeakageTestA.AlarmTime.PT:= T#5s;

            SC_P3_LeakageTestA.IdleTime.IN:= TRUE;

            IF SC_P3_LeakageTestA.IdleTime.Q THEN
                SC_P3_LeakageTestA.ResetStep:= TRUE;
                SC_P3_LeakageTestA.Step:= 3;
            END_IF

        3:
            SC_P3_LeakageTestA.StepName:='3 - Inicializacia - zasunutie pritlaku';
            SC_P3_LeakageTestA.IdleTime.PT:= T#2s;
            SC_P3_LeakageTestA.AlarmTime.PT:= T#5s;

            IF NOT SC_P3_LeakageTestA.Switch1 THEN
                P3_LeakageTestA.OUT.PneuZamok_ODOMKNI_YV159:= TRUE;
                Pritlak_ZASUN:= TRUE;
                SC_P3_LeakageTestA.Switch1:= TRUE;
            END_IF

            IF P3_LeakageTestA.IN.Pritlak_ZASUNUTY_MS46 THEN
                P3_LeakageTestA.OUT.PneuZamok_ODOMKNI_YV159:= FALSE;
                SC_P3_LeakageTestA.ResetStep:= TRUE;
                SC_P3_LeakageTestA.Step:= 8;
            END_IF

        8:
            SC_P3_LeakageTestA.StepName:='8 - Inicializacia - zasunutie centrovacky';
            SC_P3_LeakageTestA.IdleTime.PT:= T#4s;
            SC_P3_LeakageTestA.AlarmTime.PT:= T#5s;

            IF NOT SC_P3_LeakageTestA.Switch1 THEN
                Centrovacku_ZASUN:= TRUE;
                SC_P3_LeakageTestA.Switch1:= TRUE;
            END_IF

            IF P3_LeakageTestA.IN.Centrovanie_ZASUNUTE_IS72 AND P3_Dopravniky.STAV.PoINIT THEN
                SC_P3_LeakageTestA.ResetStep:= TRUE;
                SC_P3_LeakageTestA.Step:= 10;
            END_IF

        10:
            SC_P3_LeakageTestA.StepName:='10 - Inicializacia - kontrola typu zalozeneho kopita';
            SC_P3_LeakageTestA.IdleTime.PT:= T#4s;
            SC_P3_LeakageTestA.AlarmTime.PT:= T#5s;

            IF Linka.PAR.ZvolenyModel = '4F' AND P3_LeakageTestA.IN.PritomnostKopita_IS67 AND P3_LeakageTestA.IN.Tester_TypKonektoru_4F THEN
                SC_P3_LeakageTestA.ResetStep:= TRUE;
                SC_P3_LeakageTestA.Step:= 13;
            ELSIF Linka.PAR.ZvolenyModel = '5F' AND P3_LeakageTestA.IN.PritomnostKopita_IS67 AND P3_LeakageTestA.IN.Tester_TypKonektoru_5F_5H THEN
                SC_P3_LeakageTestA.ResetStep:= TRUE;
                SC_P3_LeakageTestA.Step:= 13;
            ELSIF Linka.PAR.ZvolenyModel = '5H' AND P3_LeakageTestA.IN.PritomnostKopita_IS67 AND P3_LeakageTestA.IN.Tester_TypKonektoru_5F_5H THEN
                SC_P3_LeakageTestA.ResetStep:= TRUE;
                SC_P3_LeakageTestA.Step:= 13;
            ELSE
                P34_Alarmy[314]:= TRUE;
                P3_PoruchaST2:= TRUE;
            END_IF

        13:
            SC_P3_LeakageTestA.StepName:='13 - Inicializacia - hladanie paletky';
            SC_P3_LeakageTestA.IdleTime.PT:= T#5s;
            SC_P3_LeakageTestA.AlarmTime.PT:= T#5s;
            SC_P3_LeakageTestA.IdleTime.IN:= TRUE;

            IF P3_LeakageTestA.IN.PritomnostPaletky_S23 THEN
                P3_AkumulacnyStoper.STAV.PrebiehaVyvezeniePaletky:= FALSE;
                SC_P3_LeakageTestA.ResetStep:= TRUE;
                SC_P3_LeakageTestA.Step:= 20;
            ELSIF SC_P3_LeakageTestA.IdleTime.Q THEN
                P3_LeakageTestA.STAV.PoINIT:= TRUE;
                SC_P3_LeakageTestA.ResetStep:= TRUE;
                SC_P3_LeakageTestA.Step:= 100;
            END_IF

        20:
            SC_P3_LeakageTestA.StepName:='20 - Inicializacia - precitanie cisla paletky';
            SC_P3_LeakageTestA.IdleTime.PT:= T#200ms;
            SC_P3_LeakageTestA.AlarmTime.PT:= T#5s;
            SC_P3_LeakageTestA.IdleTime.IN:= TRUE;

            IF SC_P3_LeakageTestA.IdleTime.Q THEN
                PrecitaneCisloPaletky:= USINT_TO_STRING(P3_LeakageTestA.IN.PrecitaneCisloPaletky_S23);
                i:= 0;
                SC_P3_LeakageTestA.ResetStep:= TRUE;
                SC_P3_LeakageTestA.Step:= 23;
            END_IF

        23:
            SC_P3_LeakageTestA.StepName:='23 - Inicializacia - priradenie indexu paletky na zaklade precitanej hodnoty';
            SC_P3_LeakageTestA.IdleTime.PT:= T#200ms;
            SC_P3_LeakageTestA.AlarmTime.PT:= T#5s;

            IF PrecitaneCisloPaletky = '171' THEN
                i:= 1;
            ELSIF PrecitaneCisloPaletky = '164' THEN
                i:= 2;
            ELSIF PrecitaneCisloPaletky = '181' THEN
                i:= 3;
            ELSIF PrecitaneCisloPaletky = '168' THEN
                i:= 4;
            ELSIF PrecitaneCisloPaletky = '140' THEN
                i:= 5;
            ELSIF PrecitaneCisloPaletky = '110' THEN
                i:= 6;
            ELSIF PrecitaneCisloPaletky = '156' THEN
                i:= 7;
            ELSIF PrecitaneCisloPaletky = '127' THEN
                i:= 8;
            ELSIF PrecitaneCisloPaletky = '139' THEN
                i:= 9;
            ELSIF PrecitaneCisloPaletky = '131' THEN
                i:= 10;
            ELSIF PrecitaneCisloPaletky = '178' THEN
                i:= 11;
            ELSIF PrecitaneCisloPaletky = '206' THEN
                i:= 12;
            ELSIF PrecitaneCisloPaletky = '119' THEN
                i:= 13;
            ELSIF PrecitaneCisloPaletky = '163' THEN
                i:= 14;
            ELSIF PrecitaneCisloPaletky = '128' THEN
                i:= 15;
            ELSIF PrecitaneCisloPaletky = '175' THEN
                i:= 16;
            ELSIF PrecitaneCisloPaletky = '138' THEN
                i:= 17;
            ELSE
                P34_Alarmy[310]:= TRUE;
                P3_PoruchaST2:= TRUE;
            END_IF

            IF i<> 0 THEN
                Paletka[i].PAR.CisloPaletky:= USINT_TO_STRING(i);
                P3_LeakageTestA.PAR.IndexPaletky_STRING:= USINT_TO_STRING(i);
                P3_LeakageTestA.PAR.IndexPaletky:= i;
                PrecitaneCisloPaletky:= '';
                SC_P3_LeakageTestA.ResetStep:= TRUE;
                SC_P3_LeakageTestA.Step:= 30;
            END_IF

        30:
            SC_P3_LeakageTestA.StepName:='30 - Inicializacia - kontrola stavu paletky';
            SC_P3_LeakageTestA.IdleTime.PT:= T#200ms;
            SC_P3_LeakageTestA.AlarmTime.PT:= T#5s;

            IF Paletka[i].PAR.TestovaciKus AND Paletka[i].PAR.CisloTestovacejStanice = 'ST_8A,8B' THEN
                IF P3_LeakageTestA.STAV.Tester_ON THEN
                    TestovaciKus:= TRUE;
                    P3_LeakageTestA.STAV.PoINIT:= TRUE;
                    SC_P3_LeakageTestA.ResetStep:= TRUE;
                    SC_P3_LeakageTestA.Step:= 113;
                ELSE
                    P3_LeakageTestA.STAV.PoINIT:= TRUE;
                    SC_P3_LeakageTestA.ResetStep:= TRUE;
                    SC_P3_LeakageTestA.Step:= 560;
                END_IF
            ELSIF Paletka[i].PAR.TestovaciKus AND Paletka[i].PAR.CisloTestovacejStanice <> 'ST_8A,8B' THEN
                P3_LeakageTestA.STAV.PoINIT:= TRUE;
                SC_P3_LeakageTestA.ResetStep:= TRUE;
                SC_P3_LeakageTestA.Step:= 560;
            ELSIF Paletka[i].PAR.RevorkovyKus AND Paletka[i].PAR.CisloRevorkovejStanice = 'ST_8A,8B' THEN
                IF P3_LeakageTestA.STAV.Tester_ON THEN
                    Revork:= TRUE;
                    P3_LeakageTestA.STAV.PoINIT:= TRUE;
                    SC_P3_LeakageTestA.ResetStep:= TRUE;
                    SC_P3_LeakageTestA.Step:= 105;
                ELSE
                    P3_LeakageTestA.STAV.PoINIT:= TRUE;
                    SC_P3_LeakageTestA.ResetStep:= TRUE;
                    SC_P3_LeakageTestA.Step:= 560;
                END_IF
            ELSIF Paletka[i].PAR.RevorkovyKus AND Paletka[i].PAR.CisloRevorkovejStanice <> 'ST_8A,8B' THEN
                Revork:= FALSE;
                P3_LeakageTestA.STAV.PoINIT:= TRUE;
                SC_P3_LeakageTestA.ResetStep:= TRUE;
                SC_P3_LeakageTestA.Step:= 560;
            ELSIF Paletka[i].PAR.StavPaletky = 'OK' THEN
                SC_P3_LeakageTestA.ResetStep:= TRUE;
                SC_P3_LeakageTestA.Step:= 33;
            ELSIF Paletka[i].PAR.StavPaletky = 'NG' THEN
                P3_LeakageTestA.STAV.PoINIT:= TRUE;
                SC_P3_LeakageTestA.ResetStep:= TRUE;
                SC_P3_LeakageTestA.Step:= 560;
            END_IF

        33:
            SC_P3_LeakageTestA.StepName:='33 - Inicializacia - kontrola uzavretia komunikacie';
            SC_P3_LeakageTestA.IdleTime.PT:= T#200ms;
            SC_P3_LeakageTestA.AlarmTime.PT:= T#5s;

            IF Paletka[i].VnutornyStav.KomunikaciaUzavreta THEN
                P3_LeakageTestA.STAV.PoINIT:= TRUE;
                SC_P3_LeakageTestA.ResetStep:= TRUE;
                SC_P3_LeakageTestA.Step:= 560;
            ELSE
                SC_P3_LeakageTestA.ResetStep:= TRUE;
                SC_P3_LeakageTestA.Step:= 35;
            END_IF

        35:
            SC_P3_LeakageTestA.StepName:='35 - Inicializacia - kontrola otvorenia komunikacie';
            SC_P3_LeakageTestA.IdleTime.PT:= T#200ms;
            SC_P3_LeakageTestA.AlarmTime.PT:= T#5s;

            IF Paletka[i].VnutornyStav.KomunikaciaOtvorena THEN
                P3_LeakageTestA.STAV.PoINIT:= TRUE;
                SC_P3_LeakageTestA.ResetStep:= TRUE;
                SC_P3_LeakageTestA.Step:= 118;
            ELSE
                P3_LeakageTestA.STAV.PoINIT:= TRUE;
                SC_P3_LeakageTestA.ResetStep:= TRUE;
                SC_P3_LeakageTestA.Step:= 100;
            END_IF

            //********************************************************Automatický režim****************************************************************************//

        100:
            SC_P3_LeakageTestA.StepName:='100 - Automaticky Rezim - cakam na príchod paletky na stoper';
            SC_P3_LeakageTestA.IdleTime.PT:= T#200ms;
            SC_P3_LeakageTestA.AlarmTime.PT:= T#5s;

            IF P3_LeakageTestA.IN.PritomnostPaletky_S23 THEN
                P3_AkumulacnyStoper.STAV.PrebiehaVyvezeniePaletky:= FALSE;
            END_IF

            SC_P3_LeakageTestA.IdleTime.IN:= P3_LeakageTestA.IN.PritomnostPaletky_S23;

            IF EDGEPOS(P3_LeakageTestA.IN.PritomnostPaletky_S23)THEN
                IF NOT Taktime_LeakageTestA_ST8A.CMD.START_Merania_1 THEN
                    Taktime_LeakageTestA_ST8A.CMD.START_Merania_1:= TRUE;
                ELSE
                    Taktime_LeakageTestA_ST8A.CMD.ZAPIS_Hodnot_1:= TRUE;
                END_IF
            END_IF

            IF P3_LeakageTestA.KoniecCyklu THEN
                SC_P3_LeakageTestA.ResetStep:= TRUE;
                SC_P3_LeakageTestA.Step:= 0;
            ELSIF SC_P3_LeakageTestA.IdleTime.Q THEN
                SC_P3_LeakageTestA.ResetStep:= TRUE;
                SC_P3_LeakageTestA.Step:= 101;
            END_IF

        101:
            SC_P3_LeakageTestA.StepName:='101 - Automaticky Rezim - precitanie cisla paletky';
            SC_P3_LeakageTestA.IdleTime.PT:= T#500ms;
            SC_P3_LeakageTestA.AlarmTime.PT:= T#5s;
            SC_P3_LeakageTestA.IdleTime.IN:= TRUE;

            PrecitaneCisloPaletky:= USINT_TO_STRING(P3_LeakageTestA.IN.PrecitaneCisloPaletky_S23);
            i:= 0;
            SC_P3_LeakageTestA.ResetStep:= TRUE;
            SC_P3_LeakageTestA.Step:= 102;

        102:
            SC_P3_LeakageTestA.StepName:='102 - Automaticky Rezim - priradenie indexu paletky na zaklade precitanej hodnoty';
            SC_P3_LeakageTestA.IdleTime.PT:= T#200ms;
            SC_P3_LeakageTestA.AlarmTime.PT:= T#5s;

            IF PrecitaneCisloPaletky = '171' THEN
                i:= 1;
            ELSIF PrecitaneCisloPaletky = '164' THEN
                i:= 2;
            ELSIF PrecitaneCisloPaletky = '181' THEN
                i:= 3;
            ELSIF PrecitaneCisloPaletky = '168' THEN
                i:= 4;
            ELSIF PrecitaneCisloPaletky = '140' THEN
                i:= 5;
            ELSIF PrecitaneCisloPaletky = '110' THEN
                i:= 6;
            ELSIF PrecitaneCisloPaletky = '156' THEN
                i:= 7;
            ELSIF PrecitaneCisloPaletky = '127' THEN
                i:= 8;
            ELSIF PrecitaneCisloPaletky = '139' THEN
                i:= 9;
            ELSIF PrecitaneCisloPaletky = '131' THEN
                i:= 10;
            ELSIF PrecitaneCisloPaletky = '178' THEN
                i:= 11;
            ELSIF PrecitaneCisloPaletky = '206' THEN
                i:= 12;
            ELSIF PrecitaneCisloPaletky = '119' THEN
                i:= 13;
            ELSIF PrecitaneCisloPaletky = '163' THEN
                i:= 14;
            ELSIF PrecitaneCisloPaletky = '128' THEN
                i:= 15;
            ELSIF PrecitaneCisloPaletky = '175' THEN
                i:= 16;
            ELSIF PrecitaneCisloPaletky = '138' THEN
                i:= 17;
            ELSE
                P34_Alarmy[310]:= TRUE;
                P3_PoruchaST2:= TRUE;
            END_IF

            IF i<> 0 THEN
                Paletka[i].PAR.CisloPaletky:= USINT_TO_STRING(i);
                P3_LeakageTestA.PAR.IndexPaletky_STRING:= USINT_TO_STRING(i);
                P3_LeakageTestA.PAR.IndexPaletky:= i;
                PrecitaneCisloPaletky:= '';
                SC_P3_LeakageTestA.ResetStep:= TRUE;
                SC_P3_LeakageTestA.Step:= 103;
            END_IF

        103:
            SC_P3_LeakageTestA.StepName:='103 - Automaticky Rezim - kontrola stavu paletky';
            SC_P3_LeakageTestA.IdleTime.PT:= T#200ms;
            SC_P3_LeakageTestA.AlarmTime.PT:= T#5s;

            IF Paletka[i].PAR.TestovaciKus AND Paletka[i].PAR.CisloTestovacejStanice = 'ST_8A,8B' THEN
                IF P3_LeakageTestA.STAV.Tester_ON THEN
                    TestovaciKus:= TRUE;
                    SC_P3_LeakageTestA.ResetStep:= TRUE;
                    SC_P3_LeakageTestA.Step:= 113;
                ELSE
                    SC_P3_LeakageTestA.ResetStep:= TRUE;
                    SC_P3_LeakageTestA.Step:= 560;
                END_IF
            ELSIF Paletka[i].PAR.TestovaciKus AND Paletka[i].PAR.CisloTestovacejStanice <> 'ST_8A,8B' THEN
                SC_P3_LeakageTestA.ResetStep:= TRUE;
                SC_P3_LeakageTestA.Step:= 560;
            ELSIF Paletka[i].PAR.RevorkovyKus AND Paletka[i].PAR.CisloRevorkovejStanice = 'ST_8A,8B' THEN
                IF P3_LeakageTestA.STAV.Tester_ON THEN
                    Revork:= TRUE;
                    SC_P3_LeakageTestA.ResetStep:= TRUE;
                    SC_P3_LeakageTestA.Step:= 105;
                ELSE
                    SC_P3_LeakageTestA.ResetStep:= TRUE;
                    SC_P3_LeakageTestA.Step:= 560;
                END_IF
            ELSIF Paletka[i].PAR.RevorkovyKus AND Paletka[i].PAR.CisloRevorkovejStanice <> 'ST_8A,8B' THEN
                Revork:= FALSE;
                SC_P3_LeakageTestA.ResetStep:= TRUE;
                SC_P3_LeakageTestA.Step:= 560;
            ELSIF Paletka[i].PAR.StavPaletky = 'OK' AND P3_LeakageTestA.STAV.Tester_ON THEN
                SC_P3_LeakageTestA.ResetStep:= TRUE;
                SC_P3_LeakageTestA.Step:= 105;
            ELSIF Paletka[i].PAR.StavPaletky = 'OK' AND NOT P3_LeakageTestA.STAV.Tester_ON THEN
                SC_P3_LeakageTestA.ResetStep:= TRUE;
                SC_P3_LeakageTestA.Step:= 560;
            ELSIF Paletka[i].PAR.StavPaletky = 'NG' THEN
                SC_P3_LeakageTestA.ResetStep:= TRUE;
                SC_P3_LeakageTestA.Step:= 560;
            END_IF

        105:
            SC_P3_LeakageTestA.StepName:='105 - Automaticky Rezim - kontrola zapnutia testovacej stanice B';
            SC_P3_LeakageTestA.IdleTime.PT:= T#200ms;
            SC_P3_LeakageTestA.AlarmTime.PT:= T#5s;

            IF P3_LeakageTestB.STAV.Tester_ON THEN
                SC_P3_LeakageTestA.ResetStep:= TRUE;
                SC_P3_LeakageTestA.Step:= 107;
            ELSE
                SC_P3_LeakageTestA.ResetStep:= TRUE;
                SC_P3_LeakageTestA.Step:= 113;
            END_IF

        107:
            SC_P3_LeakageTestA.StepName:='107 - Automaticky Rezim - kontrola paletky v testovacej stanic1 B';
            SC_P3_LeakageTestA.IdleTime.PT:= T#1s;
            SC_P3_LeakageTestA.AlarmTime.PT:= T#5s;
            SC_P3_LeakageTestA.IdleTime.IN:= TRUE;

            IF P3_LeakageTestA.KoniecCyklu THEN
                SC_P3_LeakageTestA.ResetStep:= TRUE;
                SC_P3_LeakageTestA.Step:= 113;
            ELSIF SC_P3_LeakageTestB.Step = 100 AND NOT P3_LeakageTestB.IN.PritomnostPaletky_S24 THEN
                SC_P3_LeakageTestA.ResetStep:= TRUE;
                SC_P3_LeakageTestA.Step:= 560;
            ELSIF SC_P3_LeakageTestB.Step = 110 AND P3_LeakageTestB.IN.PritomnostPaletky_S24 THEN
                SC_P3_LeakageTestA.ResetStep:= TRUE;
                SC_P3_LeakageTestA.Step:= 110;
            END_IF

        110:
            SC_P3_LeakageTestA.StepName:='110 - Automaticky Rezim - cakam na spustenie testovania';
            SC_P3_LeakageTestA.IdleTime.PT:= T#200ms;
            SC_P3_LeakageTestA.AlarmTime.PT:= T#5s;

            IF P3_LeakageTestB.OUT.KOM_StanicaA_StartTestovania THEN
                P3_LeakageTestB.OUT.KOM_StanicaA_StartTestovania:= FALSE;
                SC_P3_LeakageTestA.ResetStep:= TRUE;
                SC_P3_LeakageTestA.Step:= 113;
            END_IF

        113:
            SC_P3_LeakageTestA.StepName:='113 - Automaticky Rezim - vyziadanie stavu paletky zo servera, zacentrovanie paletky';
            SC_P3_LeakageTestA.IdleTime.PT:= T#200ms;
            SC_P3_LeakageTestA.AlarmTime.PT:= T#5s;
            SC_P3_LeakageTestA.IdleTime.IN:= TRUE;

            IF NOT SC_P3_LeakageTestA.Switch1 THEN
                TRCB_P3_LeakageTestA_ST8A.CMD.VyziadajStavPaletky_TYP1:= TRUE;
                Centrovacku_VYSUN:= TRUE;
                SC_P3_LeakageTestA.Switch1:= TRUE;
            END_IF

            IF TRCB_P3_LeakageTestA_ST8A.STATUS.KomunikaciaUkoncena THEN
                TRCB_P3_LeakageTestA_ST8A.CMD.VyziadajStavPaletky_TYP1:= FALSE;
                SC_P3_LeakageTestA.ResetStep:= TRUE;
                SC_P3_LeakageTestA.Step:= 114;
            ELSIF TRCB_P3_LeakageTestA_ST8A.STATUS.KomunikaciaError THEN
                TRCB_P3_LeakageTestA_ST8A.CMD.VyziadajStavPaletky_TYP1:= FALSE;
                SC_P3_LeakageTestA.ResetStep:= TRUE;
                SC_P3_LeakageTestA.Step:= 115;
            END_IF

        114:
            SC_P3_LeakageTestA.StepName:='114 - Automaticky Rezim - kontrola odpovede servera';
            SC_P3_LeakageTestA.IdleTime.PT:= T#200ms;
            SC_P3_LeakageTestA.AlarmTime.PT:= T#5s;

            IF NOT TRCB_P3_LeakageTestA_ST8A.STATUS.KomunikaciaUkoncena AND P3_LeakageTestA.IN.Centrovanie_VYSUNUTE_IS71 THEN
                IF TRCB_P3_LeakageTestA_ST8A.OUTPUTS.PovolenieCinnostiNaPaletke = 'OK' THEN
                    Paletka[i].VnutornyStav.KomunikaciaOtvorena:= TRUE;
                    IF TRCB_P3_LeakageTestA_ST8A.OUTPUTS.DruhCinnostiNaPaletke  = 'PRD;ST8A' THEN
                        SC_P3_LeakageTestA.ResetStep:= TRUE;
                        SC_P3_LeakageTestA.Step:= 118;
                    ELSIF TRCB_P3_LeakageTestA_ST8A.OUTPUTS.DruhCinnostiNaPaletke  = 'SMP;ST8A,ST8B' THEN
                        SC_P3_LeakageTestA.ResetStep:= TRUE;
                        SC_P3_LeakageTestA.Step:= 118;
                    ELSIF TRCB_P3_LeakageTestA_ST8A.OUTPUTS.DruhCinnostiNaPaletke  = 'PRD;ST8A,ST8B' THEN
                        SC_P3_LeakageTestA.ResetStep:= TRUE;
                        SC_P3_LeakageTestA.Step:= 118;
                    ELSE
                        Paletka[i].PAR.StavPaletky := 'NG';
                        SC_P3_LeakageTestA.ResetStep:= TRUE;
                        SC_P3_LeakageTestA.Step:= 116;
                    END_IF
                ELSIF TRCB_P3_LeakageTestA_ST8A.OUTPUTS.PovolenieCinnostiNaPaletke = 'NG' THEN
                    SC_P3_LeakageTestA.ResetStep:= TRUE;
                    SC_P3_LeakageTestA.Step:= 115;
                END_IF
            END_IF

        115:
            SC_P3_LeakageTestA.StepName:='115 - Automaticky Rezim - rozhodnutie obsluhy po odpovedi panatrace NG';
            SC_P3_LeakageTestA.IdleTime.PT:= T#200ms;
            SC_P3_LeakageTestA.AlarmTime.PT:= T#5s;

            P34_Vizu.ZobrazHL1_ST8:= TRUE;

            IF TRCB_P3_LeakTestA_OpatovnyDopyt THEN
                TRCB_P3_LeakTestA_OpatovnyDopyt:= FALSE;
                P34_Vizu.ZobrazHL1_ST8:= FALSE;
                SC_P3_LeakageTestA.ResetStep:= TRUE;
                SC_P3_LeakageTestA.Step:= 113;
            ELSIF TRCB_P3_LeakTestA_PaletkaNG THEN
                TRCB_P3_LeakTestA_PaletkaNG:= FALSE;
                P34_Vizu.ZobrazHL1_ST8:= FALSE;
                Paletka[i].PAR.StavPaletky := 'NG';
                SC_P3_LeakageTestA.ResetStep:= TRUE;
                SC_P3_LeakageTestA.Step:= 116;
            END_IF

        116:
            SC_P3_LeakageTestA.StepName:='116 - Automaticky Rezim - odcentrovanie paletky po odpovedi servera NG';
            SC_P3_LeakageTestA.IdleTime.PT:= T#200ms;
            SC_P3_LeakageTestA.AlarmTime.PT:= T#5s;

            IF NOT SC_P3_LeakageTestA.Switch1 THEN
                Centrovacku_ZASUN:= TRUE;
                SC_P3_LeakageTestA.Switch1:= TRUE;
            END_IF

            IF P3_LeakageTestA.IN.Centrovanie_ZASUNUTE_IS72 THEN
                SC_P3_LeakageTestA.ResetStep:= TRUE;
                SC_P3_LeakageTestA.Step:= 560;
            END_IF

        118:
            SC_P3_LeakageTestA.StepName:='118 - Automaticky Rezim - zacentrovanie paletky ';
            SC_P3_LeakageTestA.IdleTime.PT:= T#200ms;
            SC_P3_LeakageTestA.AlarmTime.PT:= T#5s;

            IF NOT SC_P3_LeakageTestA.Switch1 THEN
                Centrovacku_VYSUN:= TRUE;
                SC_P3_LeakageTestA.Switch1:= TRUE;
            END_IF

            IF P3_LeakageTestA.IN.Centrovanie_VYSUNUTE_IS71 THEN
                SC_P3_LeakageTestA.ResetStep:= TRUE;
                SC_P3_LeakageTestA.Step:= 120;
            END_IF

        120:
            SC_P3_LeakageTestA.StepName:='120 - Automaticky Rezim - vysunutie horneho pritlaku ';
            SC_P3_LeakageTestA.IdleTime.PT:= T#3s;
            SC_P3_LeakageTestA.AlarmTime.PT:= T#5s;

            IF NOT SC_P3_LeakageTestA.Switch1 THEN
                P3_LeakageTestA.OUT.PneuZamok_ODOMKNI_YV159:= TRUE;
                Pritlak_VYSUN:= TRUE;
                SC_P3_LeakageTestA.Switch1:= TRUE;
            END_IF

            IF P3_LeakageTestA.IN.Pritlak_VYSUNUTY_MS47 THEN
                SC_P3_LeakageTestA.ResetStep:= TRUE;
                SC_P3_LeakageTestA.Step:= 123;
            END_IF

        123:
            SC_P3_LeakageTestA.StepName:='123 - Automaticky Rezim - vysunutie spodneho kopita';
            SC_P3_LeakageTestA.IdleTime.PT:= T#1s;
            SC_P3_LeakageTestA.AlarmTime.PT:= T#5s;
            SC_P3_LeakageTestA.IdleTime.IN:= TRUE;

            IF P3_LeakageTestA.IN.PritomnostKopita_IS67 AND P3_LeakageTestA.IN.Kopito_ZASUNUTE_IS68 THEN
                P3_LeakageTestA.OUT.Kopito_ZASUN_YV142:= FALSE;
                P3_LeakageTestA.OUT.Kopito_VYSUN_YV141:= TRUE;
                SC_P3_LeakageTestA.ResetStep:= TRUE;
                SC_P3_LeakageTestA.Step:= 125;
            END_IF

        125:
            SC_P3_LeakageTestA.StepName:='125 - Automaticky Rezim - cakam na spustenie testera';
            SC_P3_LeakageTestA.IdleTime.PT:= T#200ms;
            SC_P3_LeakageTestA.AlarmTime.PT:= T#300ms;

            SC_P3_LeakageTestA.IdleTime.IN:= NOT P3_LeakageTestA.IN.Kopito_ZASUNUTE_IS68;

            IF SC_P3_LeakageTestA.IdleTime.Q THEN
                SC_P3_LeakageTestA.ResetStep:= TRUE;
                SC_P3_LeakageTestA.Step:= 130;
            END_IF

        130:
            SC_P3_LeakageTestA.StepName:='130 - Automaticky Rezim - spustenie testera';
            SC_P3_LeakageTestA.IdleTime.PT:= T#4s800ms;
            SC_P3_LeakageTestA.AlarmTime.PT:= T#5s;

            IF NOT SC_P3_LeakageTestA.Switch1 AND AteqLeakageTester_A.Stav_READY THEN
                AteqLeakageTester_A.START_Testovania:= TRUE;
                Paletka[i].VnutornyStav.CinnostSpustena:= TRUE;
                SC_P3_LeakageTestA.IdleTime.IN:= TRUE;
                SC_P3_LeakageTestA.Switch1:= TRUE;
            END_IF

            IF NOT AteqLeakageTester_A.Stav_READY AND AteqLeakageTester_A.Stav_START_DONE AND NOT AteqLeakageTester_A.VysledokTestovania_OK AND NOT AteqLeakageTester_A.VysledokTestovania_NG AND SC_P3_LeakageTestA.IdleTime.Q THEN
                P3_LeakageTestA.OUT.PneuZamok_ODOMKNI_YV159:= FALSE;
                P3_LeakageTestA.OUT.Pritlak_VYSUN_YV157:= FALSE;
                SC_P3_LeakageTestA.ResetStep:= TRUE;
                SC_P3_LeakageTestA.Step:= 133;
            END_IF

        133:
            SC_P3_LeakageTestA.StepName:='130 - Automaticky Rezim - nacitanie parametrov testera';
            SC_P3_LeakageTestA.IdleTime.PT:= T#500ms;
            SC_P3_LeakageTestA.AlarmTime.PT:= T#5s;

            IF AteqLeakageTester_A.Stav_READY THEN
                AteqLeakageTester_A.START_Testovania:= FALSE;
                AteqLeakageTester_A.CitajParametreTestera:= TRUE;
            END_IF

            SC_P3_LeakageTestA.IdleTime.IN:= AteqLeakageTester_A.Stav_CitanieParametrov_OK;

            IF AteqLeakageTester_A.Stav_CitanieParametrov_OK AND SC_P3_LeakageTestA.IdleTime.Q THEN
                Reports.LeakageTest.CasPlnenia.StanicaA:= REAL_TO_STRING(AteqLeakageTester_A.CasPnenia);
                Reports.LeakageTest.CasStabilizacie.StanicaA:= REAL_TO_STRING(AteqLeakageTester_A.CasStabilizacie);
                Reports.LeakageTest.TlakPlnenia.StanicaA:= REAL_TO_STRING(AteqLeakageTester_A.TlakPlnenia);
                Reports.LeakageTest.ToleranciaPritlaku_MIN.StanicaA:= '';
                Reports.LeakageTest.ToleranciaPritlaku_MAX.StanicaA:= '';
                Reports.LeakageTest.TlakPritlaku.StanicaA:= REAL_TO_STRING(P3_LeakageTestA.IN.PreratanyVyrovnavaciTlak_Bar);
                Reports.LeakageTest.TlakUniku.StanicaA:= REAL_TO_STRING(AteqLeakageTester_A.TlakUniku);
                Reports.LeakageTest.ToleranciaTlakUniku_MIN.StanicaA:= REAL_TO_STRING(AteqLeakageTester_A.Tolerancia * -1);
                Reports.LeakageTest.ToleranciaTlakUniku_MAX.StanicaA:= REAL_TO_STRING(AteqLeakageTester_A.Tolerancia);
                Reports.LeakageTest.Tolerancia.StanicaA:= REAL_TO_STRING(AteqLeakageTester_A.Tolerancia);
                AteqLeakageTester_A.CitajParametreTestera:= FALSE;
                SC_P3_LeakageTestA.ResetStep:= TRUE;
                SC_P3_LeakageTestA.Step:= 135;
            END_IF

        135:
            SC_P3_LeakageTestA.StepName:='135 - Automaticky Rezim - kontrola výsledku testu';
            SC_P3_LeakageTestA.IdleTime.PT:= T#1s;
            SC_P3_LeakageTestA.AlarmTime.PT:= T#5s;

            IF AteqLeakageTester_A.VysledokTestovania_OK THEN
                Paletka[i].VnutornyStav.LeakageTest_Ukonceny:= TRUE;
                Reports.LeakageTest.VyslednyReport.StanicaA:= 'PASS';
                Paletka[i].PAR.StavPowerCP:= 'PASS';
                Paletka[i].VnutornyStav.CinnostUkoncena:= TRUE;
                SC_P3_LeakageTestA.ResetStep:= TRUE;
                SC_P3_LeakageTestA.Step:= 140;
            ELSE
                IF NOT Revork THEN
                    OpakovanyTest:= TRUE;
                END_IF
                Paletka[i].PAR.StavPowerCP:= 'FAIL';
                Paletka[i].VnutornyStav.CinnostUkoncena:= TRUE;
                Reports.LeakageTest.VyslednyReport.StanicaA:= 'FAIL';
                SC_P3_LeakageTestA.ResetStep:= TRUE;
                SC_P3_LeakageTestA.Step:= 140;
            END_IF

        140:
            SC_P3_LeakageTestA.StepName:='140 - Automaticky Rezim - cakam na ukoncenie testovania testera stanice B';
            SC_P3_LeakageTestA.IdleTime.PT:= T#1s;
            SC_P3_LeakageTestA.AlarmTime.PT:= T#5s;

            IF NOT AteqLeakageTester_B.START_Testovania THEN
                SC_P3_LeakageTestA.ResetStep:= TRUE;
                SC_P3_LeakageTestA.Step:= 150;
            ELSIF P3_LeakageTestA.RR_TestovaciaSekvencia THEN
                SC_P3_LeakageTestA.ResetStep:= TRUE;
                SC_P3_LeakageTestA.Step:= 150;
            END_IF

        150:
            SC_P3_LeakageTestA.StepName:='150 - Automaticky Rezim - zasunutie spodneho kopita ';
            SC_P3_LeakageTestA.IdleTime.PT:= T#200ms;
            SC_P3_LeakageTestA.AlarmTime.PT:= T#5s;

            P3_LeakageTestA.OUT.Kopito_VYSUN_YV141:= FALSE;
            P3_LeakageTestA.OUT.Kopito_ZASUN_YV142:= TRUE;

            IF P3_LeakageTestA.IN.Kopito_ZASUNUTE_IS68 THEN
                SC_P3_LeakageTestA.ResetStep:= TRUE;
                SC_P3_LeakageTestA.Step:= 153;
            END_IF

        153:
            SC_P3_LeakageTestA.StepName:='153 - Automaticky Rezim - zasunutie horneho pritlaku';
            SC_P3_LeakageTestA.IdleTime.PT:= T#200ms;
            SC_P3_LeakageTestA.AlarmTime.PT:= T#5s;

            IF NOT SC_P3_LeakageTestA.Switch1 THEN
                P3_LeakageTestA.OUT.PneuZamok_ODOMKNI_YV159:= TRUE;
                Pritlak_ZASUN:= TRUE;
                SC_P3_LeakageTestA.IdleTime.IN:= TRUE;
                SC_P3_LeakageTestA.Switch1:= TRUE;
            END_IF

            IF SC_P3_LeakageTestA.IdleTime.Q THEN
                SC_P3_LeakageTestA.ResetStep:= TRUE;
                SC_P3_LeakageTestA.Step:= 545;
            END_IF

            //Odcentrovanie paletky//

        545:
            SC_P3_LeakageTestA.StepName:='545 - Automaticky Rezim - odcentrovanie paletky';
            SC_P3_LeakageTestA.IdleTime.PT:= T#200ms;
            SC_P3_LeakageTestA.AlarmTime.PT:= T#5s;

            Centrovacku_ZASUN:= TRUE;
            IF P3_LeakageTestA.RR_TestovaciaSekvencia THEN
                SC_P3_LeakageTestA.ResetStep:= TRUE;
                SC_P3_LeakageTestA.Step:= 558;
            ELSE
                SC_P3_LeakageTestA.ResetStep:= TRUE;
                SC_P3_LeakageTestA.Step:= 550;
            END_IF

            //Odoslanie dát na server//

        550:
            SC_P3_LeakageTestA.StepName:='550 - Automaticky Rezim - odoslanie stavu paletky na server';
            SC_P3_LeakageTestA.IdleTime.PT:= T#200ms;
            SC_P3_LeakageTestA.AlarmTime.PT:= T#5s;

            IF NOT SC_P3_LeakageTestA.Switch1 THEN
                TRCB_P3_LeakageTestA_ST8A.CMD.OdosliStavPaletky_TYP2:= TRUE;
                SC_P3_LeakageTestA.Switch1:= TRUE;
            END_IF

            IF TRCB_P3_LeakageTestA_ST8A.STATUS.KomunikaciaUkoncena THEN
                TRCB_P3_LeakageTestA_ST8A.CMD.OdosliStavPaletky_TYP2:= FALSE;
                SC_P3_LeakageTestA.ResetStep:= TRUE;
                SC_P3_LeakageTestA.Step:= 553;
            ELSIF TRCB_P3_LeakageTestA_ST8A.STATUS.KomunikaciaError THEN
                //                P34_Alarmy[311]:= TRUE;
                //                P3_PoruchaST2:= TRUE;
            END_IF

        553:
            SC_P3_LeakageTestA.StepName:='553 - Automaticky Rezim - kontrola odpovede servera';
            SC_P3_LeakageTestA.IdleTime.PT:= T#200ms;
            SC_P3_LeakageTestA.AlarmTime.PT:= T#5s;

            IF NOT TRCB_P3_LeakageTestA_ST8A.STATUS.KomunikaciaUkoncena THEN
                IF TRCB_P3_LeakageTestA_ST8A.OUTPUTS.PovolenieCinnostiNaPaletke = 'OK' THEN
                    Paletka[i].PAR.StavPaletky:= 'OK';
                    SC_P3_LeakageTestA.ResetStep:= TRUE;
                    SC_P3_LeakageTestA.Step:= 554;
                ELSIF TRCB_P3_LeakageTestA_ST8A.OUTPUTS.PovolenieCinnostiNaPaletke = 'NG' THEN
                    Paletka[i].PAR.StavPaletky:= 'NG';
                    SC_P3_LeakageTestA.ResetStep:= TRUE;
                    SC_P3_LeakageTestA.Step:= 554;
                END_IF
            END_IF

        554:
            SC_P3_LeakageTestA.StepName:='554 - Automaticky Rezim - kontrola poctu testovani';
            SC_P3_LeakageTestA.IdleTime.PT:= T#1s;
            SC_P3_LeakageTestA.AlarmTime.PT:= T#5s;
            SC_P3_LeakageTestA.IdleTime.IN:= TRUE;

            IF NOT SC_P3_LeakageTestA.Switch1 THEN
                PocetOpakovaniTestu:= PocetOpakovaniTestu + 1;
                SC_P3_LeakageTestA.Switch1:= TRUE;
            END_IF

            IF OpakovanyTest AND PocetOpakovaniTestu < 2 AND SC_P3_LeakageTestA.IdleTime.Q AND NOT TestovaciKus THEN
                OpakovanyTest:= FALSE;
                SC_P3_LeakageTestA.ResetStep:= TRUE;
                SC_P3_LeakageTestA.Step:= 113;
            ELSIF OpakovanyTest AND PocetOpakovaniTestu >= 2 AND NOT TestovaciKus THEN
                Paletka[i].VnutornyStav.LeakageTest_Ukonceny:= TRUE;
                OpakovanyTest:= FALSE;
                PocetOpakovaniTestu:= 0;
                SC_P3_LeakageTestA.ResetStep:= TRUE;
                SC_P3_LeakageTestA.Step:= 555;
            ELSIF NOT OpakovanyTest OR TestovaciKus THEN
                SC_P3_LeakageTestA.ResetStep:= TRUE;
                SC_P3_LeakageTestA.Step:= 555;
            END_IF

        555:
            SC_P3_LeakageTestA.StepName:='555 - Automaticky Rezim - vyhodnotenie stavu paletky';
            SC_P3_LeakageTestA.IdleTime.PT:= T#200ms;
            SC_P3_LeakageTestA.AlarmTime.PT:= T#5s;

            IF Paletka[i].PAR.StavPaletky = 'OK' THEN
                IF Paletka[i].PAR.StavPowerCP = 'PASS' THEN
                    Paletka[i].PAR.StavPaletky:= 'OK';
                ELSIF Paletka[i].PAR.StavPowerCP = 'FAIL' THEN
                    Paletka[i].PAR.StavPaletky:= 'NG';
                END_IF
            END_IF
            Paletka[i].VnutornyStav.KomunikaciaUzavreta:= TRUE;

            SC_P3_LeakageTestA.ResetStep:= TRUE;
            SC_P3_LeakageTestA.Step:= 558;

        558:
            SC_P3_LeakageTestA.StepName:='558 - Automaticky Rezim - kontrola otvorenia testera';
            SC_P3_LeakageTestA.IdleTime.PT:= T#200ms;
            SC_P3_LeakageTestA.AlarmTime.PT:= T#5s;

            IF P3_LeakageTestA.IN.Centrovanie_ZASUNUTE_IS72 AND P3_LeakageTestA.IN.Pritlak_ZASUNUTY_MS46 AND P3_LeakageTestA.IN.Kopito_ZASUNUTE_IS68 THEN
                P3_LeakageTestA.OUT.PneuZamok_ODOMKNI_YV159:= FALSE;
                IF P3_LeakageTestA.RR_TestovaciaSekvencia THEN
                    P3_LeakageTestA.RR_TestovaciaSekvencia:= FALSE;
                    SC_P3_LeakageTestA.ResetStep:= TRUE;
                    SC_P3_LeakageTestA.Step:= 700;
                ELSE
                    SC_P3_LeakageTestA.ResetStep:= TRUE;
                    SC_P3_LeakageTestA.Step:= 560;
                END_IF
            END_IF

            //Vyvezenie paletky//

        560:
            SC_P3_LeakageTestA.StepName:='560 - Automaticky Rezim - cakam na vyvezenie na stoper leakage testu B';
            SC_P3_LeakageTestA.IdleTime.PT:= T#200ms;
            SC_P3_LeakageTestA.AlarmTime.PT:= T#5s;

            IF P3_LeakageTestA.KoniecCyklu THEN
                SC_P3_LeakageTestA.ResetStep:= TRUE;
                SC_P3_LeakageTestA.Step:= 0;
            ELSIF ((NOT P3_LeakageTestB.IN.PritomnostPaletky_S24 AND SC_P3_LeakageTestB.Step = 100) OR (P3_LeakageTestB.OUT.ZasunStoper_YV135 AND SC_P3_LeakageTestB.Step = 561)) AND NOT P3_LeakageTestA.STAV.PrebiehaVyvezeniePaletky AND NOT TEST THEN
                P3_LeakageTestA.OUT.ZasunStoper_YV134:= TRUE;
                P3_LeakageTestA.STAV.PrebiehaVyvezeniePaletky:= TRUE;
                SC_P3_LeakageTestA.ResetStep:= TRUE;
                SC_P3_LeakageTestA.Step:= 561;
            END_IF

        561:
            SC_P3_LeakageTestA.StepName:='561 - Automaticky Rezim - ukoncenie vyvazania na stoper leakage testu B';
            SC_P3_LeakageTestA.IdleTime.PT:= T#200ms;
            SC_P3_LeakageTestA.AlarmTime.PT:= T#10s;

            SC_P3_LeakageTestA.IdleTime.IN:= NOT P3_LeakageTestA.IN.PritomnostPaletky_S23;
            SC_P3_LeakageTestA.AlarmTime.IN:= P3_LeakageTestA.IN.PritomnostPaletky_S23;

            IF NOT P3_LeakageTestA.IN.PritomnostPaletky_S23 THEN
                IF Revork THEN
                    Paletka[i].PAR.RevorkovyKus:= FALSE;
                    Paletka[i].PAR.CisloRevorkovejStanice:= '';
                    Revork:= FALSE;
                END_IF
                P3_LeakageTestA.OUT.ZasunStoper_YV134:= FALSE;
                TestovaciKus:= FALSE;
                OpakovanyTest:= FALSE;
                PocetOpakovaniTestu:= 0;
                Paletka[i].PAR.StavPowerCP:= '';
                Paletka[i].VnutornyStav.CinnostSpustena:= FALSE;
                Paletka[i].VnutornyStav.CinnostUkoncena:= FALSE;
                Paletka[i].VnutornyStav.FotkyOdoslane:= FALSE;
                Paletka[i].VnutornyStav.KomunikaciaOtvorena:= FALSE;
                Paletka[i].VnutornyStav.KomunikaciaUzavreta:= FALSE;
                Reports.LeakageTest.CasPlnenia.StanicaA:= '';
                Reports.LeakageTest.VyslednyReport.StanicaA:= '';
                Reports.LeakageTest.CasStabilizacie.StanicaA:= '';
                Reports.LeakageTest.TlakPlnenia.StanicaA:= '';
                Reports.LeakageTest.ToleranciaPritlaku_MIN.StanicaA:= '';
                Reports.LeakageTest.ToleranciaPritlaku_MAX.StanicaA:= '';
                Reports.LeakageTest.TlakPritlaku.StanicaA:= '';
                Reports.LeakageTest.TlakUniku.StanicaA:= '';
                Reports.LeakageTest.Tolerancia.StanicaA:= '';
            END_IF

            IF SC_P3_LeakageTestA.IdleTime.Q AND NOT P3_LeakageTestA.OUT.ZasunStoper_YV134 THEN
                SC_P3_LeakageTestA.ResetStep:= TRUE;
                SC_P3_LeakageTestA.Step:= 100;
            ELSIF SC_P3_LeakageTestA.AlarmTime.Q THEN
                P34_Alarmy[357]:= TRUE;
                P3_Pracovisko.KoniecCyklu:= TRUE;
                SC_P3_LeakageTestA.ResetStep:= TRUE;
                SC_P3_LeakageTestA.Step:= 0;
            END_IF

            //*******************************************************Manuálny režim*******************************************************************************//
        700:
            SC_P3_LeakageTestA.StepName:='700 - Manualny Rezim';
            SC_P3_LeakageTestA.IdleTime.PT:= T#8s;
            SC_P3_LeakageTestA.AlarmTime.PT:= T#5s;

            P3_LeakageTestA.OUT.PneuZamok_ODOMKNI_YV159:= TRUE;

            //Vysunutie spodného kopita//
            IF P3_LeakageTestA.RR_VysunSpodneKopito THEN
                P3_LeakageTestA.OUT.Kopito_ZASUN_YV142:= FALSE;
                P3_LeakageTestA.OUT.Kopito_VYSUN_YV141:= TRUE;
            ELSE
                P3_LeakageTestA.OUT.Kopito_VYSUN_YV141:= FALSE;
                P3_LeakageTestA.OUT.Kopito_ZASUN_YV142:= TRUE;
            END_IF

            //Spustenie testovacej sekvencie//
            P3_LeakageTestA.STAV.TestovaciaSekvencia_BUSY:= P3_LeakageTestA.RR_TestovaciaSekvencia;

            IF P3_LeakageTestA.RR_TestovaciaSekvencia THEN
                IF P3_LeakageTestA.IN.PritomnostPaletky_S23 THEN
                    SC_P3_LeakageTestA.ResetStep:= TRUE;
                    SC_P3_LeakageTestA.Step:= 118;
                ELSE
                    P3_LeakageTestA.RR_TestovaciaSekvencia:= FALSE;
                END_IF
            END_IF

    END_CASE

				END_PROGRAM

PROGRAM _EXIT
				(* Insert code here *)

				END_PROGRAM
```

#### Variables.var - Local variables
```iecst
VAR
	SC_OvlCentrovacky : SequenceControlTyp;
	Centrovacku_VYSUN : BOOL;
	Centrovacku_ZASUN : BOOL;
	PrecitaneCisloPaletky : STRING[3];
	ServerOdpoved_StavPowerCP : STRING[5];
	i : USINT;
	SC_OvlPritlaku : SequenceControlTyp;
	Pritlak_VYSUN : BOOL;
	Pritlak_ZASUN : BOOL;
	TEST : BOOL;
	IdentifikaciaParametra1 : USINT;
	IdentifikaciaParametra2 : USINT;
	IdentifikaciaParametra3 : USINT;
	IdentifikaciaParametra4 : USINT;
	PocetCitanychParametrov : USINT;
	PocetDopytovNaServer : USINT;
	CasPneniaREAL : REAL;
	CasStabilizacieREAL : REAL;
	TlakPlneniaREAL : REAL;
	ToleranciaREAL : REAL;
	TlakUnikuREAL : REAL;
	PaletkaPrechadza : BOOL;
	TestovaciKus : BOOL;
	Revork : BOOL;
	Triger_0 : BOOL;
	Triger_1 : BOOL;
	PocetOpakovaniTestu : USINT;
	OpakovanyTest : BOOL;
END_VAR
```

#### IOLinkKomunikacia.st
```iecst
ACTION IOLinkKomunikacia:

	//Snímač paletky//
	P3_LeakageTestA.IN.PritomnostPaletky_S23:= P3_LeakageTestA.PAR.SnimacPaletky_IOLinkInputs[1].0;
	P3_LeakageTestA.IN.PrecitaneCisloPaletky_S23:= P3_LeakageTestA.PAR.SnimacPaletky_IOLinkInputs[9];

	//Snímač tlaku//
	P3_LeakageTestA.IN.VyrovnavaciTlak_OK_S26:= P3_LeakageTestA.PAR.SnimacTlaku_IOLinkInputs.0;

	P3_LeakageTestA.IN.PrecitanyVyrovnavaciTlak_S26.0:= P3_LeakageTestA.PAR.SnimacTlaku_IOLinkInputs.2;
	P3_LeakageTestA.IN.PrecitanyVyrovnavaciTlak_S26.1:= P3_LeakageTestA.PAR.SnimacTlaku_IOLinkInputs.3;
	P3_LeakageTestA.IN.PrecitanyVyrovnavaciTlak_S26.2:= P3_LeakageTestA.PAR.SnimacTlaku_IOLinkInputs.4;
	P3_LeakageTestA.IN.PrecitanyVyrovnavaciTlak_S26.3:= P3_LeakageTestA.PAR.SnimacTlaku_IOLinkInputs.5;
	P3_LeakageTestA.IN.PrecitanyVyrovnavaciTlak_S26.4:= P3_LeakageTestA.PAR.SnimacTlaku_IOLinkInputs.6;
	P3_LeakageTestA.IN.PrecitanyVyrovnavaciTlak_S26.5:= P3_LeakageTestA.PAR.SnimacTlaku_IOLinkInputs.7;
	P3_LeakageTestA.IN.PrecitanyVyrovnavaciTlak_S26.6:= P3_LeakageTestA.PAR.SnimacTlaku_IOLinkInputs.8;
	P3_LeakageTestA.IN.PrecitanyVyrovnavaciTlak_S26.7:= P3_LeakageTestA.PAR.SnimacTlaku_IOLinkInputs.9;
	P3_LeakageTestA.IN.PrecitanyVyrovnavaciTlak_S26.8:= P3_LeakageTestA.PAR.SnimacTlaku_IOLinkInputs.10;
	P3_LeakageTestA.IN.PrecitanyVyrovnavaciTlak_S26.9:= P3_LeakageTestA.PAR.SnimacTlaku_IOLinkInputs.11;
	P3_LeakageTestA.IN.PrecitanyVyrovnavaciTlak_S26.10:= P3_LeakageTestA.PAR.SnimacTlaku_IOLinkInputs.12;
	P3_LeakageTestA.IN.PrecitanyVyrovnavaciTlak_S26.11:= P3_LeakageTestA.PAR.SnimacTlaku_IOLinkInputs.13;
	P3_LeakageTestA.IN.PrecitanyVyrovnavaciTlak_S26.12:= P3_LeakageTestA.PAR.SnimacTlaku_IOLinkInputs.14;
	P3_LeakageTestA.IN.PrecitanyVyrovnavaciTlak_S26.13:= P3_LeakageTestA.PAR.SnimacTlaku_IOLinkInputs.15;

	P3_LeakageTestA.IN.PreratanyVyrovnavaciTlak_Bar:= P3_LeakageTestA.IN.PrecitanyVyrovnavaciTlak_S26 * 0.1;

END_ACTION
```

#### OvlCentrovacky.st
```iecst
ACTION OvlCentrovacky:

	//Volanie funkcie SequenceControl//
	SequenceControl(SC:= SC_OvlCentrovacky);

	CASE SC_OvlCentrovacky.Step OF

		0:
			SC_OvlCentrovacky.StepName:= '0 - Nulovanie';
			Centrovacku_VYSUN:= FALSE;
			Centrovacku_ZASUN:= FALSE;
			P3_LeakageTestA.OUT.VysunCentrovanie_YV143:= FALSE;
			P3_LeakageTestA.OUT.ZasunCentrovanie_YV144:= FALSE;

			IF SC_P3_LeakageTestA.Step <> 0 THEN
				SC_OvlCentrovacky.ResetStep:= TRUE;
				SC_OvlCentrovacky.Step:= 1;
			END_IF

		1:
			SC_OvlCentrovacky.StepName:= '1 - Rozhodnutie o cinnosti';
			IF Centrovacku_VYSUN THEN
				SC_OvlCentrovacky.Step:= 10;
			ELSIF Centrovacku_ZASUN THEN
				SC_OvlCentrovacky.Step:= 20;
			END_IF

		10:
			SC_OvlCentrovacky.StepName:= '10 - Vysunutie centrovacky';
			SC_OvlCentrovacky.IdleTime.PT:= T#3s;
			SC_OvlCentrovacky.AlarmTime.PT:= T#30s;

			IF P3_LeakageTestA.Automat THEN
				SC_OvlCentrovacky.AlarmTime.IN:= TRUE;
			ELSE
				SC_OvlCentrovacky.IdleTime.IN:= TRUE;
			END_IF

			IF NOT SC_OvlCentrovacky.Switch1 THEN
				P3_LeakageTestA.OUT.ZasunCentrovanie_YV144:= FALSE;
				P3_LeakageTestA.OUT.VysunCentrovanie_YV143:= TRUE;
				SC_OvlCentrovacky.Switch1:= TRUE;
			END_IF

            IF P3_LeakageTestA.IN.Centrovanie_VYSUNUTE_IS71 THEN
                SC_OvlCentrovacky.IdleTime.IN:= TRUE;
            END_IF

			IF SC_OvlCentrovacky.IdleTime.Q THEN
				SC_OvlCentrovacky.ResetStep:= TRUE;
				SC_OvlCentrovacky.Step:= 0;
			ELSIF SC_OvlCentrovacky.AlarmTime.Q THEN
				P34_Alarmy[302]:= TRUE;
				P3_PoruchaST2:= TRUE;
			END_IF

		20:
			SC_OvlCentrovacky.StepName:= '20 - Zasunutie centrovacky';
			SC_OvlCentrovacky.IdleTime.PT:= T#3s;
			SC_OvlCentrovacky.AlarmTime.PT:= T#30s;

			IF P3_LeakageTestA.Automat THEN
				SC_OvlCentrovacky.AlarmTime.IN:= TRUE;
			ELSE
				SC_OvlCentrovacky.IdleTime.IN:= TRUE;
			END_IF

			IF NOT SC_OvlCentrovacky.Switch1 THEN
				P3_LeakageTestA.OUT.VysunCentrovanie_YV143:= FALSE;
				P3_LeakageTestA.OUT.ZasunCentrovanie_YV144:= TRUE;
				SC_OvlCentrovacky.Switch1:= TRUE;
			END_IF

			IF P3_LeakageTestA.IN.Centrovanie_ZASUNUTE_IS72 OR SC_OvlCentrovacky.IdleTime.Q THEN
				SC_OvlCentrovacky.ResetStep:= TRUE;
				SC_OvlCentrovacky.Step:= 0;
			ELSIF SC_OvlCentrovacky.AlarmTime.Q THEN
				P34_Alarmy[303]:= TRUE;
				P3_PoruchaST2:= TRUE;
			END_IF

	END_CASE

END_ACTION
```

#### OvlPritlaku.st
```iecst
ACTION OvlPritlaku:

	//Volanie funkcie SequenceControl//
	SequenceControl(SC:= SC_OvlPritlaku);

	CASE SC_OvlPritlaku.Step OF

		0:
			SC_OvlPritlaku.StepName:= '0 - Nulovanie';
			Pritlak_VYSUN:= FALSE;
			Pritlak_ZASUN:= FALSE;
			(*P3_LeakageTestA.OUT.Pritlak_VYSUN_YV157:= FALSE;*)
			P3_LeakageTestA.OUT.Pritlak_ZASUN_YV158:= FALSE;

			IF SC_P3_LeakageTestA.Step <> 0 THEN
				SC_OvlPritlaku.ResetStep:= TRUE;
				SC_OvlPritlaku.Step:= 1;
			END_IF

		1:
			SC_OvlPritlaku.StepName:= '1 - Rozhodnutie o cinnosti';
			IF Pritlak_VYSUN THEN
				SC_OvlPritlaku.Step:= 10;
			ELSIF Pritlak_ZASUN THEN
				SC_OvlPritlaku.Step:= 20;
			END_IF

		10:
			SC_OvlPritlaku.StepName:= '10 - Vysunutie pritlaku';
			SC_OvlPritlaku.IdleTime.PT:= T#3s;
			SC_OvlPritlaku.AlarmTime.PT:= T#30s;

			IF P3_LeakageTestA.Automat THEN
				SC_OvlPritlaku.AlarmTime.IN:= TRUE;
			ELSE
				SC_OvlPritlaku.IdleTime.IN:= TRUE;
			END_IF

			IF NOT SC_OvlPritlaku.Switch1 THEN
				P3_LeakageTestA.OUT.Pritlak_ZASUN_YV158:= FALSE;
				P3_LeakageTestA.OUT.Pritlak_VYSUN_YV157:= TRUE;
				SC_OvlPritlaku.Switch1:= TRUE;
			END_IF

			IF P3_LeakageTestA.IN.Pritlak_VYSUNUTY_MS47 OR SC_OvlPritlaku.IdleTime.Q THEN
				SC_OvlPritlaku.ResetStep:= TRUE;
				SC_OvlPritlaku.Step:= 0;
			ELSIF SC_OvlPritlaku.AlarmTime.Q THEN
				P34_Alarmy[306]:= TRUE;
				P3_PoruchaST2:= TRUE;
			END_IF

		20:
			SC_OvlPritlaku.StepName:= '20 - Zasunutie pritlaku';
			SC_OvlPritlaku.IdleTime.PT:= T#3s;
			SC_OvlPritlaku.AlarmTime.PT:= T#30s;

			IF P3_LeakageTestA.Automat THEN
				SC_OvlPritlaku.AlarmTime.IN:= TRUE;
			ELSE
				SC_OvlPritlaku.IdleTime.IN:= TRUE;
			END_IF

			IF NOT SC_OvlPritlaku.Switch1 THEN
				P3_LeakageTestA.OUT.Pritlak_VYSUN_YV157:= FALSE;
				P3_LeakageTestA.OUT.Pritlak_ZASUN_YV158:= TRUE;
				SC_OvlPritlaku.Switch1:= TRUE;
			END_IF

			IF P3_LeakageTestA.IN.Pritlak_ZASUNUTY_MS46 OR SC_OvlPritlaku.IdleTime.Q THEN
				SC_OvlPritlaku.ResetStep:= TRUE;
				SC_OvlPritlaku.Step:= 0;
			ELSIF SC_OvlPritlaku.AlarmTime.Q THEN
				P34_Alarmy[307]:= TRUE;
				P3_PoruchaST2:= TRUE;
			END_IF

	END_CASE

END_ACTION
```
